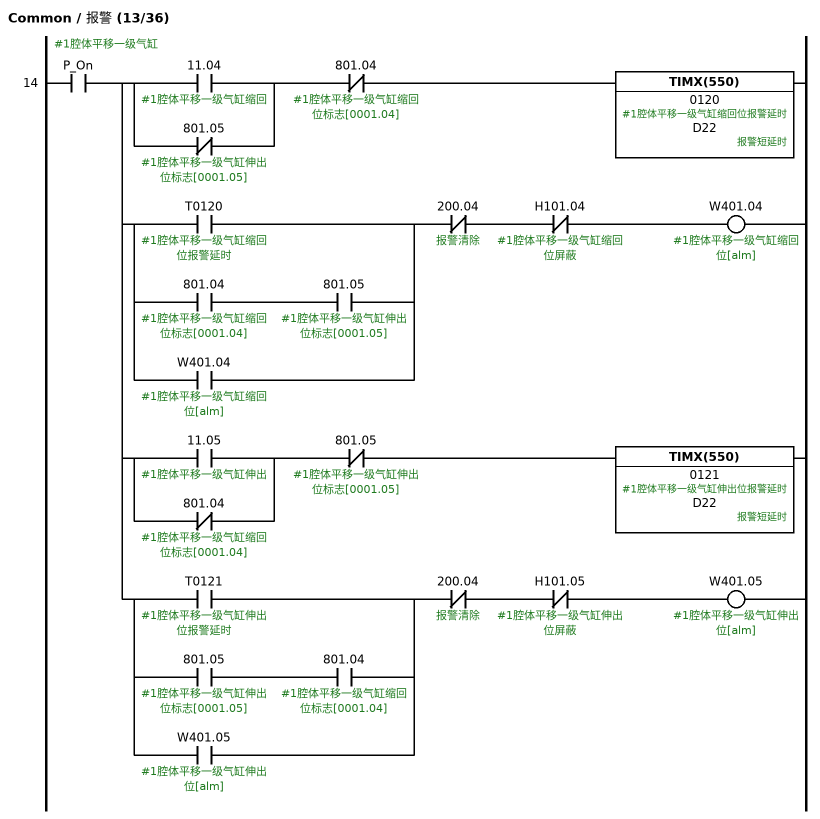
; [picture p528: Common / 报警, rungs 14-14]
; rung 14: #1腔体平移一级气缸
LD P_On
OUT TR0
LD 11.04  ; #1腔体平移一级气缸缩回
ORNOT 801.05  ; #1腔体平移一级气缸伸出位标志[0001.05]
ANDLD
ANDNOT 801.04  ; #1腔体平移一级气缸缩回位标志[0001.04]
TIMX(550) 0120 D22  ; 报警短延时, #1腔体平移一级气缸缩回位报警延时
LD TR0
LD T0120  ; #1腔体平移一级气缸缩回位报警延时
LD 801.04  ; #1腔体平移一级气缸缩回位标志[0001.04]
AND 801.05  ; #1腔体平移一级气缸伸出位标志[0001.05]
ORLD
OR W401.04  ; #1腔体平移一级气缸缩回位[alm]
ANDLD
ANDNOT 200.04  ; 报警清除
ANDNOT H101.04  ; #1腔体平移一级气缸缩回位屏蔽
OUT W401.04  ; #1腔体平移一级气缸缩回位[alm]
LD TR0
LD 11.05  ; #1腔体平移一级气缸伸出
ORNOT 801.04  ; #1腔体平移一级气缸缩回位标志[0001.04]
ANDLD
ANDNOT 801.05  ; #1腔体平移一级气缸伸出位标志[0001.05]
TIMX(550) 0121 D22  ; 报警短延时, #1腔体平移一级气缸伸出位报警延时
LD TR0
LD T0121  ; #1腔体平移一级气缸伸出位报警延时
LD 801.05  ; #1腔体平移一级气缸伸出位标志[0001.05]
AND 801.04  ; #1腔体平移一级气缸缩回位标志[0001.04]
ORLD
OR W401.05  ; #1腔体平移一级气缸伸出位[alm]
ANDLD
ANDNOT 200.04  ; 报警清除
ANDNOT H101.05  ; #1腔体平移一级气缸伸出位屏蔽
OUT W401.05  ; #1腔体平移一级气缸伸出位[alm]

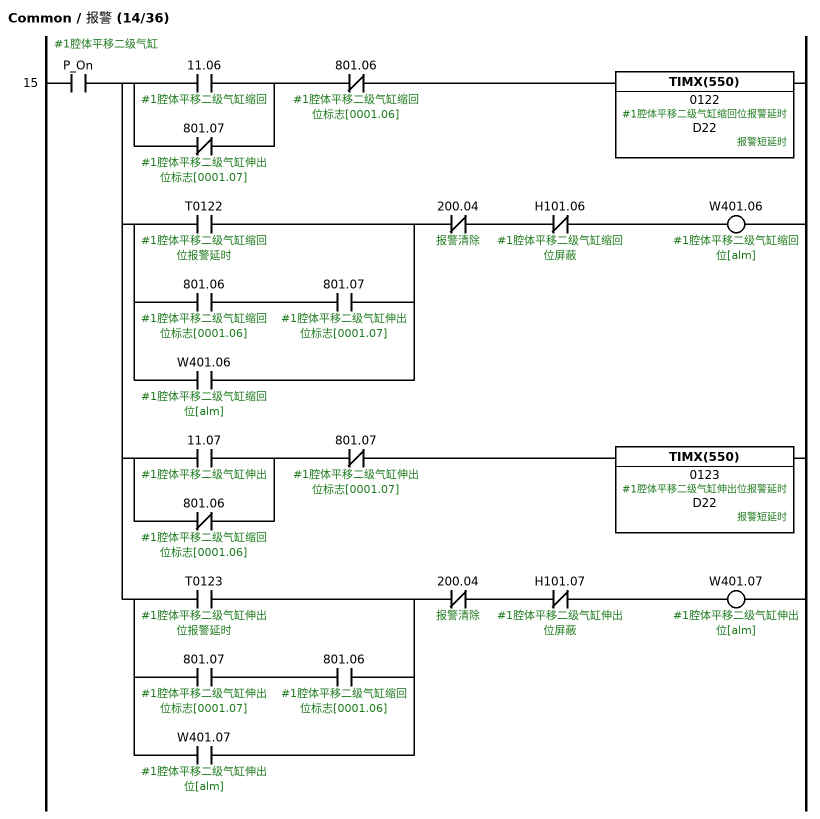
; rung 15: #1腔体平移二级气缸
LD P_On
OUT TR0
LD 11.06  ; #1腔体平移二级气缸缩回
ORNOT 801.07  ; #1腔体平移二级气缸伸出位标志[0001.07]
ANDLD
ANDNOT 801.06  ; #1腔体平移二级气缸缩回位标志[0001.06]
TIMX(550) 0122 D22  ; 报警短延时, #1腔体平移二级气缸缩回位报警延时
LD TR0
LD T0122  ; #1腔体平移二级气缸缩回位报警延时
LD 801.06  ; #1腔体平移二级气缸缩回位标志[0001.06]
AND 801.07  ; #1腔体平移二级气缸伸出位标志[0001.07]
ORLD
OR W401.06  ; #1腔体平移二级气缸缩回位[alm]
ANDLD
ANDNOT 200.04  ; 报警清除
ANDNOT H101.06  ; #1腔体平移二级气缸缩回位屏蔽
OUT W401.06  ; #1腔体平移二级气缸缩回位[alm]
LD TR0
LD 11.07  ; #1腔体平移二级气缸伸出
ORNOT 801.06  ; #1腔体平移二级气缸缩回位标志[0001.06]
ANDLD
ANDNOT 801.07  ; #1腔体平移二级气缸伸出位标志[0001.07]
TIMX(550) 0123 D22  ; 报警短延时, #1腔体平移二级气缸伸出位报警延时
LD TR0
LD T0123  ; #1腔体平移二级气缸伸出位报警延时
LD 801.07  ; #1腔体平移二级气缸伸出位标志[0001.07]
AND 801.06  ; #1腔体平移二级气缸缩回位标志[0001.06]
ORLD
OR W401.07  ; #1腔体平移二级气缸伸出位[alm]
ANDLD
ANDNOT 200.04  ; 报警清除
ANDNOT H101.07  ; #1腔体平移二级气缸伸出位屏蔽
OUT W401.07  ; #1腔体平移二级气缸伸出位[alm]

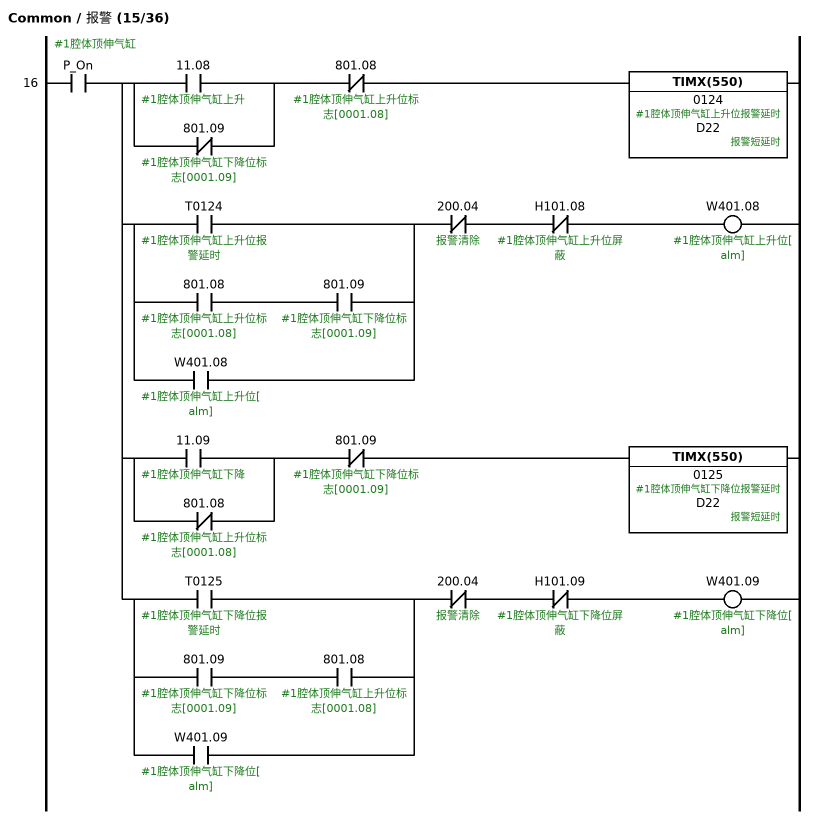
; rung 16: #1腔体顶伸气缸
LD P_On
OUT TR0
LD 11.08  ; #1腔体顶伸气缸上升
ORNOT 801.09  ; #1腔体顶伸气缸下降位标志[0001.09]
ANDLD
ANDNOT 801.08  ; #1腔体顶伸气缸上升位标志[0001.08]
TIMX(550) 0124 D22  ; 报警短延时, #1腔体顶伸气缸上升位报警延时
LD TR0
LD T0124  ; #1腔体顶伸气缸上升位报警延时
LD 801.08  ; #1腔体顶伸气缸上升位标志[0001.08]
AND 801.09  ; #1腔体顶伸气缸下降位标志[0001.09]
ORLD
OR W401.08  ; #1腔体顶伸气缸上升位[alm]
ANDLD
ANDNOT 200.04  ; 报警清除
ANDNOT H101.08  ; #1腔体顶伸气缸上升位屏蔽
OUT W401.08  ; #1腔体顶伸气缸上升位[alm]
LD TR0
LD 11.09  ; #1腔体顶伸气缸下降
ORNOT 801.08  ; #1腔体顶伸气缸上升位标志[0001.08]
ANDLD
ANDNOT 801.09  ; #1腔体顶伸气缸下降位标志[0001.09]
TIMX(550) 0125 D22  ; 报警短延时, #1腔体顶伸气缸下降位报警延时
LD TR0
LD T0125  ; #1腔体顶伸气缸下降位报警延时
LD 801.09  ; #1腔体顶伸气缸下降位标志[0001.09]
AND 801.08  ; #1腔体顶伸气缸上升位标志[0001.08]
ORLD
OR W401.09  ; #1腔体顶伸气缸下降位[alm]
ANDLD
ANDNOT 200.04  ; 报警清除
ANDNOT H101.09  ; #1腔体顶伸气缸下降位屏蔽
OUT W401.09  ; #1腔体顶伸气缸下降位[alm]

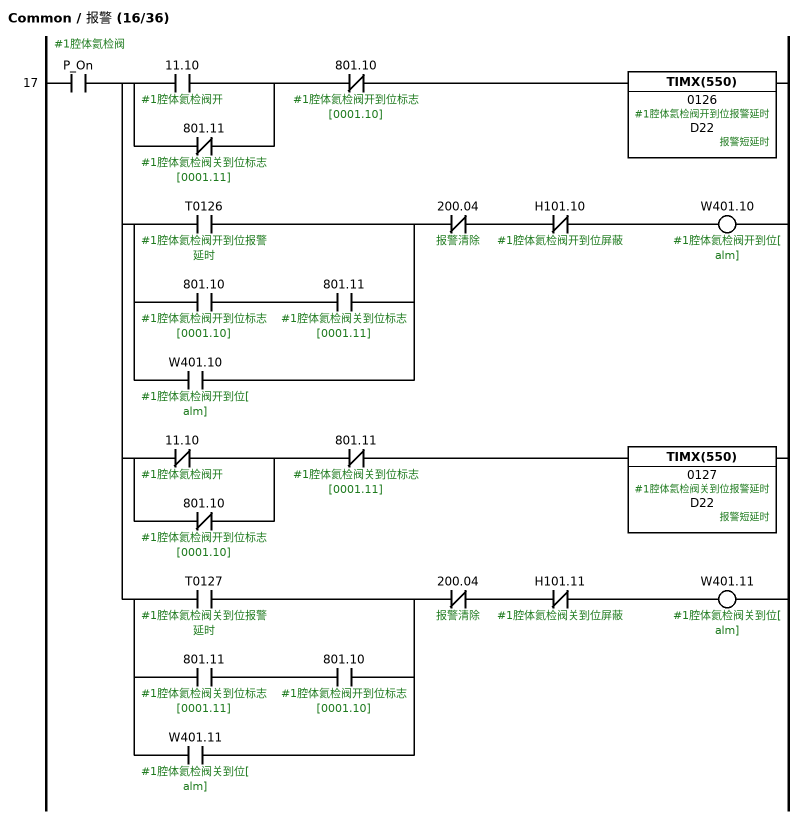
; rung 17: #1腔体氦检阀
LD P_On
OUT TR0
LD 11.10  ; #1腔体氦检阀开
ORNOT 801.11  ; #1腔体氦检阀关到位标志[0001.11]
ANDLD
ANDNOT 801.10  ; #1腔体氦检阀开到位标志[0001.10]
TIMX(550) 0126 D22  ; 报警短延时, #1腔体氦检阀开到位报警延时
LD TR0
LD T0126  ; #1腔体氦检阀开到位报警延时
LD 801.10  ; #1腔体氦检阀开到位标志[0001.10]
AND 801.11  ; #1腔体氦检阀关到位标志[0001.11]
ORLD
OR W401.10  ; #1腔体氦检阀开到位[alm]
ANDLD
ANDNOT 200.04  ; 报警清除
ANDNOT H101.10  ; #1腔体氦检阀开到位屏蔽
OUT W401.10  ; #1腔体氦检阀开到位[alm]
LD TR0
LDNOT 11.10  ; #1腔体氦检阀开
ORNOT 801.10  ; #1腔体氦检阀开到位标志[0001.10]
ANDLD
ANDNOT 801.11  ; #1腔体氦检阀关到位标志[0001.11]
TIMX(550) 0127 D22  ; 报警短延时, #1腔体氦检阀关到位报警延时
LD TR0
LD T0127  ; #1腔体氦检阀关到位报警延时
LD 801.11  ; #1腔体氦检阀关到位标志[0001.11]
AND 801.10  ; #1腔体氦检阀开到位标志[0001.10]
ORLD
OR W401.11  ; #1腔体氦检阀关到位[alm]
ANDLD
ANDNOT 200.04  ; 报警清除
ANDNOT H101.11  ; #1腔体氦检阀关到位屏蔽
OUT W401.11  ; #1腔体氦检阀关到位[alm]

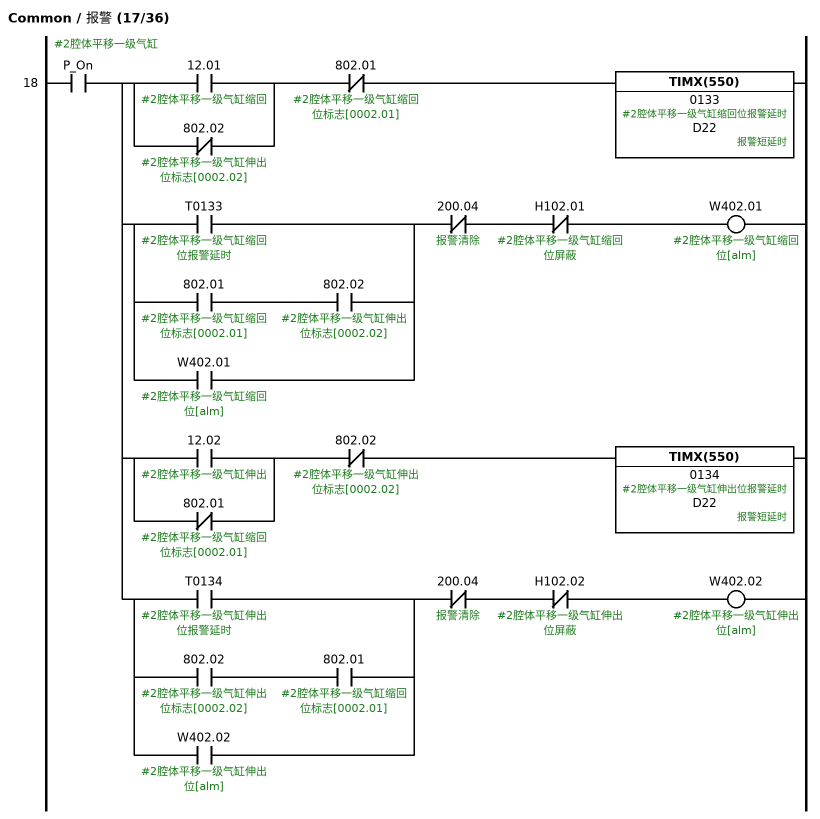
; rung 18: #2腔体平移一级气缸
LD P_On
OUT TR0
LD 12.01  ; #2腔体平移一级气缸缩回
ORNOT 802.02  ; #2腔体平移一级气缸伸出位标志[0002.02]
ANDLD
ANDNOT 802.01  ; #2腔体平移一级气缸缩回位标志[0002.01]
TIMX(550) 0133 D22  ; 报警短延时, #2腔体平移一级气缸缩回位报警延时
LD TR0
LD T0133  ; #2腔体平移一级气缸缩回位报警延时
LD 802.01  ; #2腔体平移一级气缸缩回位标志[0002.01]
AND 802.02  ; #2腔体平移一级气缸伸出位标志[0002.02]
ORLD
OR W402.01  ; #2腔体平移一级气缸缩回位[alm]
ANDLD
ANDNOT 200.04  ; 报警清除
ANDNOT H102.01  ; #2腔体平移一级气缸缩回位屏蔽
OUT W402.01  ; #2腔体平移一级气缸缩回位[alm]
LD TR0
LD 12.02  ; #2腔体平移一级气缸伸出
ORNOT 802.01  ; #2腔体平移一级气缸缩回位标志[0002.01]
ANDLD
ANDNOT 802.02  ; #2腔体平移一级气缸伸出位标志[0002.02]
TIMX(550) 0134 D22  ; 报警短延时, #2腔体平移一级气缸伸出位报警延时
LD TR0
LD T0134  ; #2腔体平移一级气缸伸出位报警延时
LD 802.02  ; #2腔体平移一级气缸伸出位标志[0002.02]
AND 802.01  ; #2腔体平移一级气缸缩回位标志[0002.01]
ORLD
OR W402.02  ; #2腔体平移一级气缸伸出位[alm]
ANDLD
ANDNOT 200.04  ; 报警清除
ANDNOT H102.02  ; #2腔体平移一级气缸伸出位屏蔽
OUT W402.02  ; #2腔体平移一级气缸伸出位[alm]

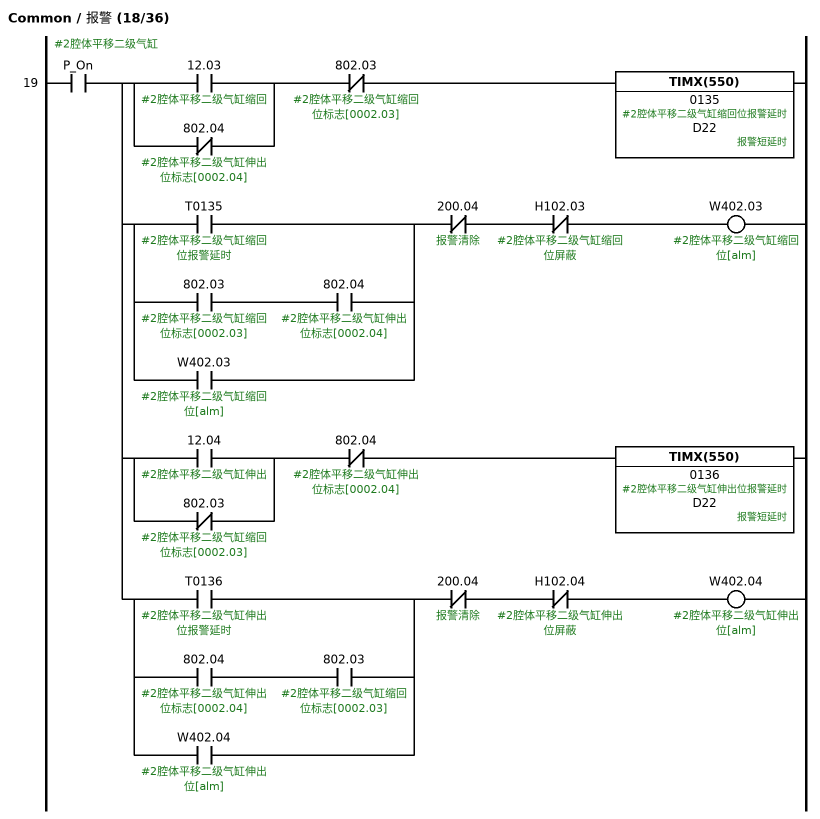
; rung 19: #2腔体平移二级气缸
LD P_On
OUT TR0
LD 12.03  ; #2腔体平移二级气缸缩回
ORNOT 802.04  ; #2腔体平移二级气缸伸出位标志[0002.04]
ANDLD
ANDNOT 802.03  ; #2腔体平移二级气缸缩回位标志[0002.03]
TIMX(550) 0135 D22  ; 报警短延时, #2腔体平移二级气缸缩回位报警延时
LD TR0
LD T0135  ; #2腔体平移二级气缸缩回位报警延时
LD 802.03  ; #2腔体平移二级气缸缩回位标志[0002.03]
AND 802.04  ; #2腔体平移二级气缸伸出位标志[0002.04]
ORLD
OR W402.03  ; #2腔体平移二级气缸缩回位[alm]
ANDLD
ANDNOT 200.04  ; 报警清除
ANDNOT H102.03  ; #2腔体平移二级气缸缩回位屏蔽
OUT W402.03  ; #2腔体平移二级气缸缩回位[alm]
LD TR0
LD 12.04  ; #2腔体平移二级气缸伸出
ORNOT 802.03  ; #2腔体平移二级气缸缩回位标志[0002.03]
ANDLD
ANDNOT 802.04  ; #2腔体平移二级气缸伸出位标志[0002.04]
TIMX(550) 0136 D22  ; 报警短延时, #2腔体平移二级气缸伸出位报警延时
LD TR0
LD T0136  ; #2腔体平移二级气缸伸出位报警延时
LD 802.04  ; #2腔体平移二级气缸伸出位标志[0002.04]
AND 802.03  ; #2腔体平移二级气缸缩回位标志[0002.03]
ORLD
OR W402.04  ; #2腔体平移二级气缸伸出位[alm]
ANDLD
ANDNOT 200.04  ; 报警清除
ANDNOT H102.04  ; #2腔体平移二级气缸伸出位屏蔽
OUT W402.04  ; #2腔体平移二级气缸伸出位[alm]

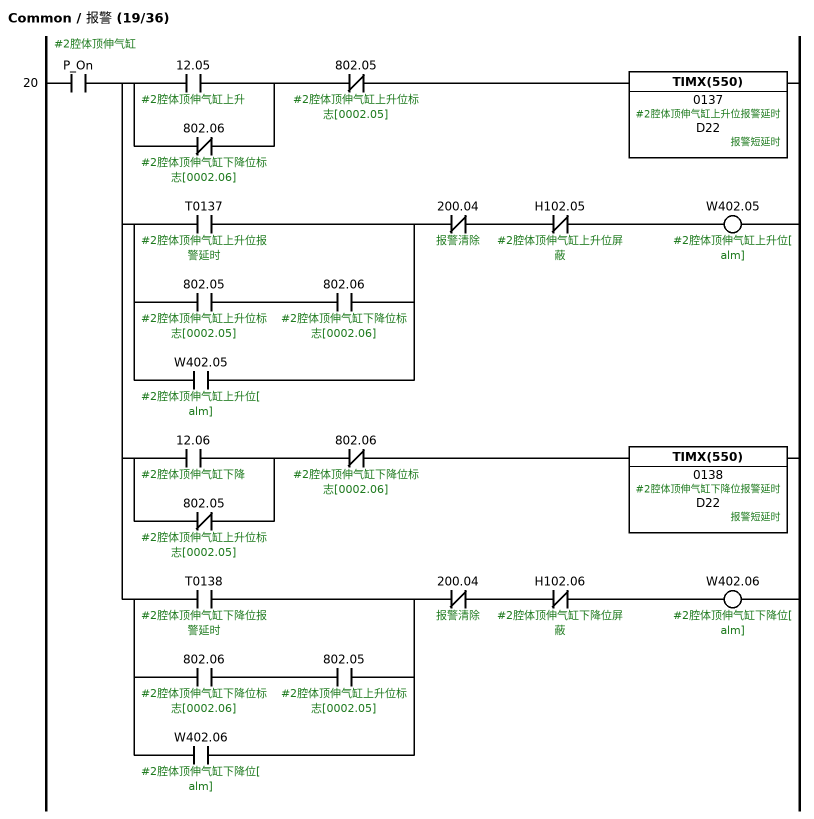
; rung 20: #2腔体顶伸气缸
LD P_On
OUT TR0
LD 12.05  ; #2腔体顶伸气缸上升
ORNOT 802.06  ; #2腔体顶伸气缸下降位标志[0002.06]
ANDLD
ANDNOT 802.05  ; #2腔体顶伸气缸上升位标志[0002.05]
TIMX(550) 0137 D22  ; 报警短延时, #2腔体顶伸气缸上升位报警延时
LD TR0
LD T0137  ; #2腔体顶伸气缸上升位报警延时
LD 802.05  ; #2腔体顶伸气缸上升位标志[0002.05]
AND 802.06  ; #2腔体顶伸气缸下降位标志[0002.06]
ORLD
OR W402.05  ; #2腔体顶伸气缸上升位[alm]
ANDLD
ANDNOT 200.04  ; 报警清除
ANDNOT H102.05  ; #2腔体顶伸气缸上升位屏蔽
OUT W402.05  ; #2腔体顶伸气缸上升位[alm]
LD TR0
LD 12.06  ; #2腔体顶伸气缸下降
ORNOT 802.05  ; #2腔体顶伸气缸上升位标志[0002.05]
ANDLD
ANDNOT 802.06  ; #2腔体顶伸气缸下降位标志[0002.06]
TIMX(550) 0138 D22  ; 报警短延时, #2腔体顶伸气缸下降位报警延时
LD TR0
LD T0138  ; #2腔体顶伸气缸下降位报警延时
LD 802.06  ; #2腔体顶伸气缸下降位标志[0002.06]
AND 802.05  ; #2腔体顶伸气缸上升位标志[0002.05]
ORLD
OR W402.06  ; #2腔体顶伸气缸下降位[alm]
ANDLD
ANDNOT 200.04  ; 报警清除
ANDNOT H102.06  ; #2腔体顶伸气缸下降位屏蔽
OUT W402.06  ; #2腔体顶伸气缸下降位[alm]

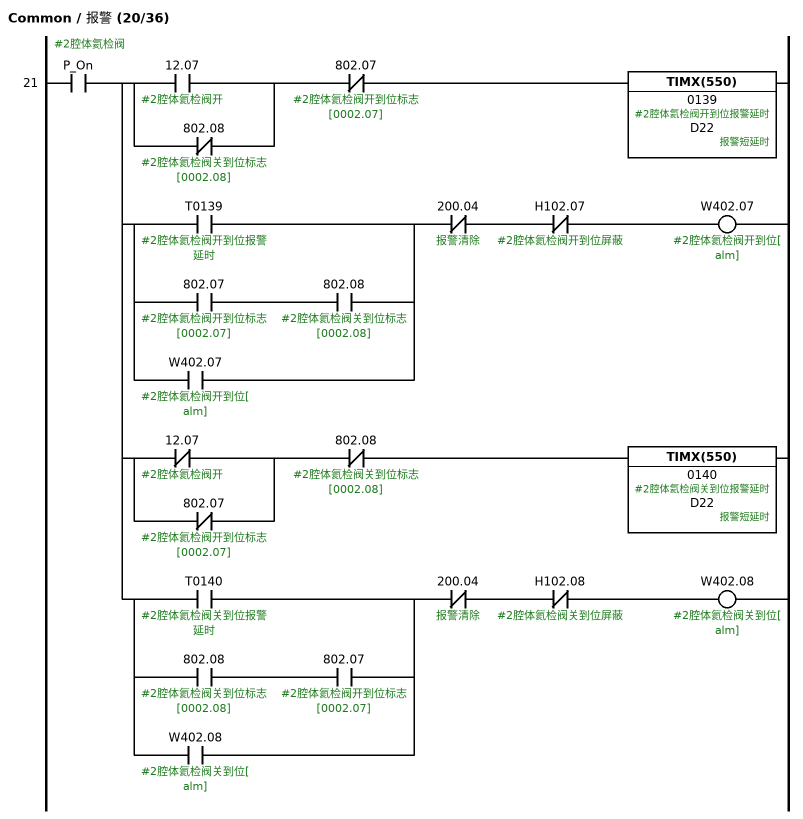
; rung 21: #2腔体氦检阀
LD P_On
OUT TR0
LD 12.07  ; #2腔体氦检阀开
ORNOT 802.08  ; #2腔体氦检阀关到位标志[0002.08]
ANDLD
ANDNOT 802.07  ; #2腔体氦检阀开到位标志[0002.07]
TIMX(550) 0139 D22  ; 报警短延时, #2腔体氦检阀开到位报警延时
LD TR0
LD T0139  ; #2腔体氦检阀开到位报警延时
LD 802.07  ; #2腔体氦检阀开到位标志[0002.07]
AND 802.08  ; #2腔体氦检阀关到位标志[0002.08]
ORLD
OR W402.07  ; #2腔体氦检阀开到位[alm]
ANDLD
ANDNOT 200.04  ; 报警清除
ANDNOT H102.07  ; #2腔体氦检阀开到位屏蔽
OUT W402.07  ; #2腔体氦检阀开到位[alm]
LD TR0
LDNOT 12.07  ; #2腔体氦检阀开
ORNOT 802.07  ; #2腔体氦检阀开到位标志[0002.07]
ANDLD
ANDNOT 802.08  ; #2腔体氦检阀关到位标志[0002.08]
TIMX(550) 0140 D22  ; 报警短延时, #2腔体氦检阀关到位报警延时
LD TR0
LD T0140  ; #2腔体氦检阀关到位报警延时
LD 802.08  ; #2腔体氦检阀关到位标志[0002.08]
AND 802.07  ; #2腔体氦检阀开到位标志[0002.07]
ORLD
OR W402.08  ; #2腔体氦检阀关到位[alm]
ANDLD
ANDNOT 200.04  ; 报警清除
ANDNOT H102.08  ; #2腔体氦检阀关到位屏蔽
OUT W402.08  ; #2腔体氦检阀关到位[alm]

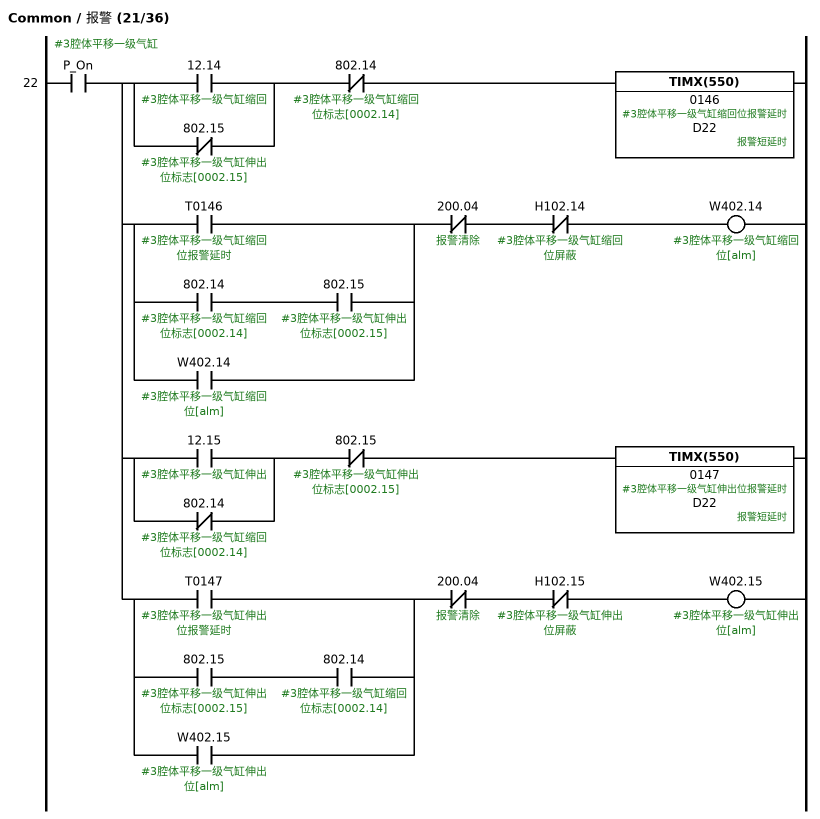
; rung 22: #3腔体平移一级气缸
LD P_On
OUT TR0
LD 12.14  ; #3腔体平移一级气缸缩回
ORNOT 802.15  ; #3腔体平移一级气缸伸出位标志[0002.15]
ANDLD
ANDNOT 802.14  ; #3腔体平移一级气缸缩回位标志[0002.14]
TIMX(550) 0146 D22  ; 报警短延时, #3腔体平移一级气缸缩回位报警延时
LD TR0
LD T0146  ; #3腔体平移一级气缸缩回位报警延时
LD 802.14  ; #3腔体平移一级气缸缩回位标志[0002.14]
AND 802.15  ; #3腔体平移一级气缸伸出位标志[0002.15]
ORLD
OR W402.14  ; #3腔体平移一级气缸缩回位[alm]
ANDLD
ANDNOT 200.04  ; 报警清除
ANDNOT H102.14  ; #3腔体平移一级气缸缩回位屏蔽
OUT W402.14  ; #3腔体平移一级气缸缩回位[alm]
LD TR0
LD 12.15  ; #3腔体平移一级气缸伸出
ORNOT 802.14  ; #3腔体平移一级气缸缩回位标志[0002.14]
ANDLD
ANDNOT 802.15  ; #3腔体平移一级气缸伸出位标志[0002.15]
TIMX(550) 0147 D22  ; 报警短延时, #3腔体平移一级气缸伸出位报警延时
LD TR0
LD T0147  ; #3腔体平移一级气缸伸出位报警延时
LD 802.15  ; #3腔体平移一级气缸伸出位标志[0002.15]
AND 802.14  ; #3腔体平移一级气缸缩回位标志[0002.14]
ORLD
OR W402.15  ; #3腔体平移一级气缸伸出位[alm]
ANDLD
ANDNOT 200.04  ; 报警清除
ANDNOT H102.15  ; #3腔体平移一级气缸伸出位屏蔽
OUT W402.15  ; #3腔体平移一级气缸伸出位[alm]

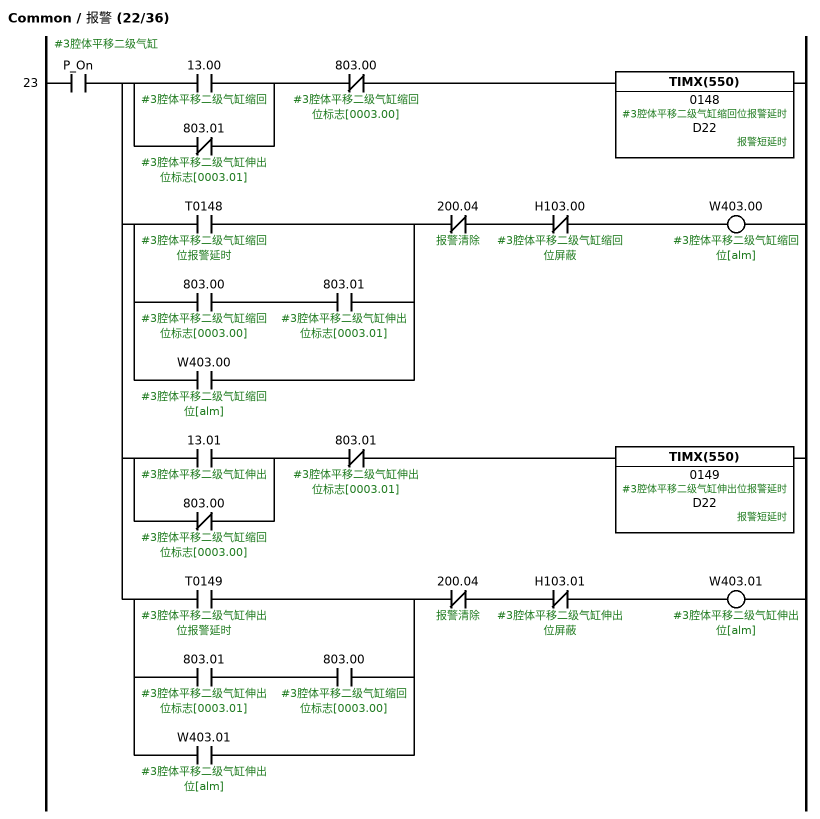
; rung 23: #3腔体平移二级气缸
LD P_On
OUT TR0
LD 13.00  ; #3腔体平移二级气缸缩回
ORNOT 803.01  ; #3腔体平移二级气缸伸出位标志[0003.01]
ANDLD
ANDNOT 803.00  ; #3腔体平移二级气缸缩回位标志[0003.00]
TIMX(550) 0148 D22  ; 报警短延时, #3腔体平移二级气缸缩回位报警延时
LD TR0
LD T0148  ; #3腔体平移二级气缸缩回位报警延时
LD 803.00  ; #3腔体平移二级气缸缩回位标志[0003.00]
AND 803.01  ; #3腔体平移二级气缸伸出位标志[0003.01]
ORLD
OR W403.00  ; #3腔体平移二级气缸缩回位[alm]
ANDLD
ANDNOT 200.04  ; 报警清除
ANDNOT H103.00  ; #3腔体平移二级气缸缩回位屏蔽
OUT W403.00  ; #3腔体平移二级气缸缩回位[alm]
LD TR0
LD 13.01  ; #3腔体平移二级气缸伸出
ORNOT 803.00  ; #3腔体平移二级气缸缩回位标志[0003.00]
ANDLD
ANDNOT 803.01  ; #3腔体平移二级气缸伸出位标志[0003.01]
TIMX(550) 0149 D22  ; 报警短延时, #3腔体平移二级气缸伸出位报警延时
LD TR0
LD T0149  ; #3腔体平移二级气缸伸出位报警延时
LD 803.01  ; #3腔体平移二级气缸伸出位标志[0003.01]
AND 803.00  ; #3腔体平移二级气缸缩回位标志[0003.00]
ORLD
OR W403.01  ; #3腔体平移二级气缸伸出位[alm]
ANDLD
ANDNOT 200.04  ; 报警清除
ANDNOT H103.01  ; #3腔体平移二级气缸伸出位屏蔽
OUT W403.01  ; #3腔体平移二级气缸伸出位[alm]

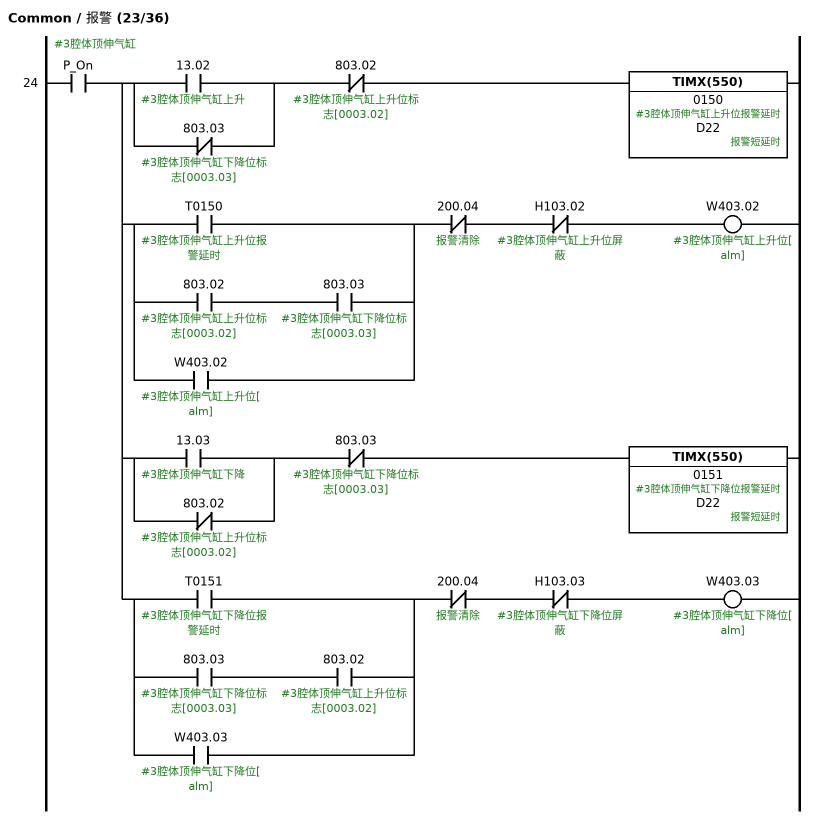
; rung 24: #3腔体顶伸气缸
LD P_On
OUT TR0
LD 13.02  ; #3腔体顶伸气缸上升
ORNOT 803.03  ; #3腔体顶伸气缸下降位标志[0003.03]
ANDLD
ANDNOT 803.02  ; #3腔体顶伸气缸上升位标志[0003.02]
TIMX(550) 0150 D22  ; 报警短延时, #3腔体顶伸气缸上升位报警延时
LD TR0
LD T0150  ; #3腔体顶伸气缸上升位报警延时
LD 803.02  ; #3腔体顶伸气缸上升位标志[0003.02]
AND 803.03  ; #3腔体顶伸气缸下降位标志[0003.03]
ORLD
OR W403.02  ; #3腔体顶伸气缸上升位[alm]
ANDLD
ANDNOT 200.04  ; 报警清除
ANDNOT H103.02  ; #3腔体顶伸气缸上升位屏蔽
OUT W403.02  ; #3腔体顶伸气缸上升位[alm]
LD TR0
LD 13.03  ; #3腔体顶伸气缸下降
ORNOT 803.02  ; #3腔体顶伸气缸上升位标志[0003.02]
ANDLD
ANDNOT 803.03  ; #3腔体顶伸气缸下降位标志[0003.03]
TIMX(550) 0151 D22  ; 报警短延时, #3腔体顶伸气缸下降位报警延时
LD TR0
LD T0151  ; #3腔体顶伸气缸下降位报警延时
LD 803.03  ; #3腔体顶伸气缸下降位标志[0003.03]
AND 803.02  ; #3腔体顶伸气缸上升位标志[0003.02]
ORLD
OR W403.03  ; #3腔体顶伸气缸下降位[alm]
ANDLD
ANDNOT 200.04  ; 报警清除
ANDNOT H103.03  ; #3腔体顶伸气缸下降位屏蔽
OUT W403.03  ; #3腔体顶伸气缸下降位[alm]

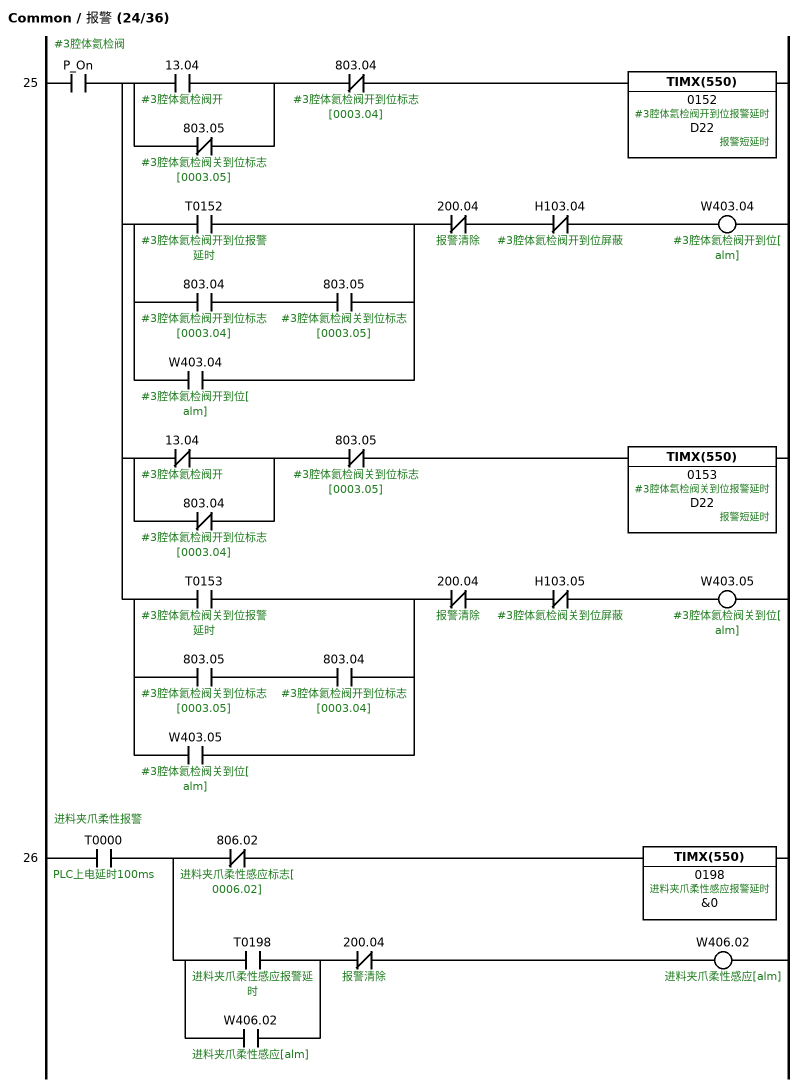
; rung 25: #3腔体氦检阀
LD P_On
OUT TR0
LD 13.04  ; #3腔体氦检阀开
ORNOT 803.05  ; #3腔体氦检阀关到位标志[0003.05]
ANDLD
ANDNOT 803.04  ; #3腔体氦检阀开到位标志[0003.04]
TIMX(550) 0152 D22  ; 报警短延时, #3腔体氦检阀开到位报警延时
LD TR0
LD T0152  ; #3腔体氦检阀开到位报警延时
LD 803.04  ; #3腔体氦检阀开到位标志[0003.04]
AND 803.05  ; #3腔体氦检阀关到位标志[0003.05]
ORLD
OR W403.04  ; #3腔体氦检阀开到位[alm]
ANDLD
ANDNOT 200.04  ; 报警清除
ANDNOT H103.04  ; #3腔体氦检阀开到位屏蔽
OUT W403.04  ; #3腔体氦检阀开到位[alm]
LD TR0
LDNOT 13.04  ; #3腔体氦检阀开
ORNOT 803.04  ; #3腔体氦检阀开到位标志[0003.04]
ANDLD
ANDNOT 803.05  ; #3腔体氦检阀关到位标志[0003.05]
TIMX(550) 0153 D22  ; 报警短延时, #3腔体氦检阀关到位报警延时
LD TR0
LD T0153  ; #3腔体氦检阀关到位报警延时
LD 803.05  ; #3腔体氦检阀关到位标志[0003.05]
AND 803.04  ; #3腔体氦检阀开到位标志[0003.04]
ORLD
OR W403.05  ; #3腔体氦检阀关到位[alm]
ANDLD
ANDNOT 200.04  ; 报警清除
ANDNOT H103.05  ; #3腔体氦检阀关到位屏蔽
OUT W403.05  ; #3腔体氦检阀关到位[alm]
; rung 26: 进料夹爪柔性报警
LD T0000  ; PLC上电延时100ms
OUT TR0
ANDNOT 806.02  ; 进料夹爪柔性感应标志[0006.02]
TIMX(550) 0198 &0  ; 进料夹爪柔性感应报警延时
LD TR0
LD T0198  ; 进料夹爪柔性感应报警延时
OR W406.02  ; 进料夹爪柔性感应[alm]
ANDLD
ANDNOT 200.04  ; 报警清除
OUT W406.02  ; 进料夹爪柔性感应[alm]

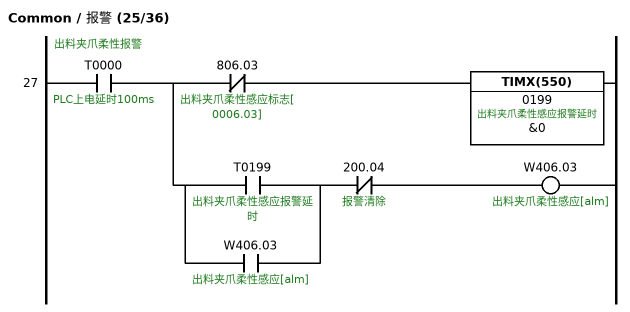
; rung 27: 出料夹爪柔性报警
LD T0000  ; PLC上电延时100ms
OUT TR0
ANDNOT 806.03  ; 出料夹爪柔性感应标志[0006.03]
TIMX(550) 0199 &0  ; 出料夹爪柔性感应报警延时
LD TR0
LD T0199  ; 出料夹爪柔性感应报警延时
OR W406.03  ; 出料夹爪柔性感应[alm]
ANDLD
ANDNOT 200.04  ; 报警清除
OUT W406.03  ; 出料夹爪柔性感应[alm]

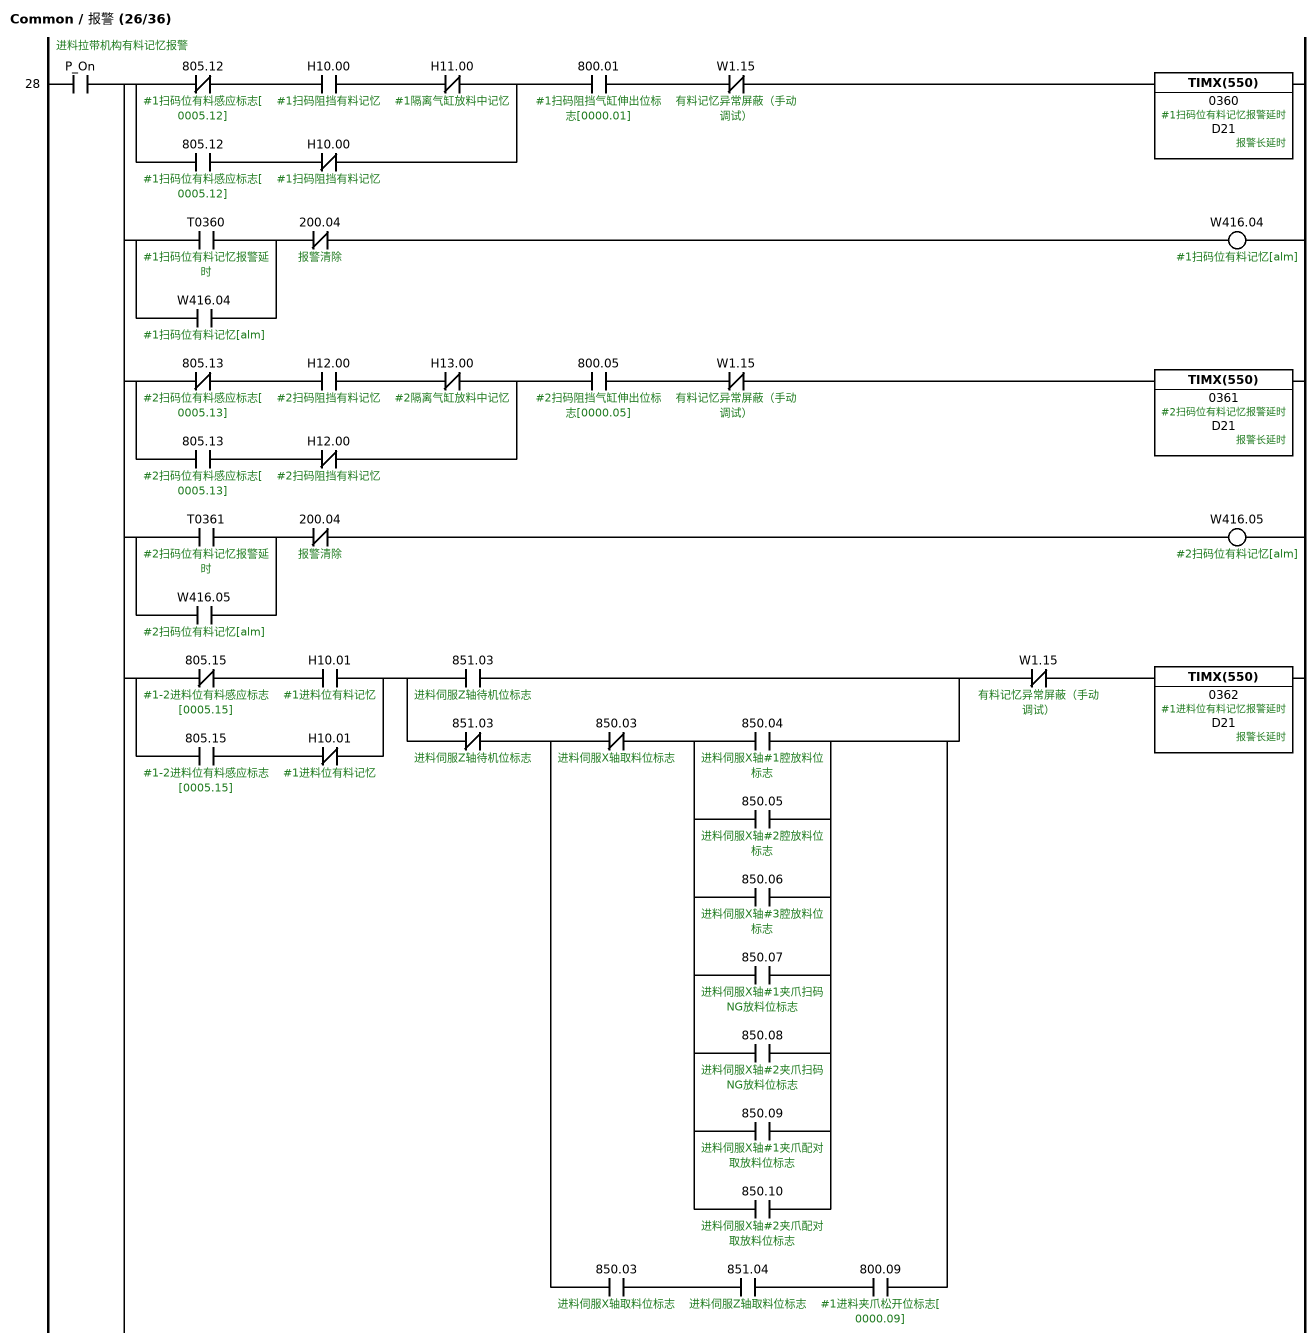

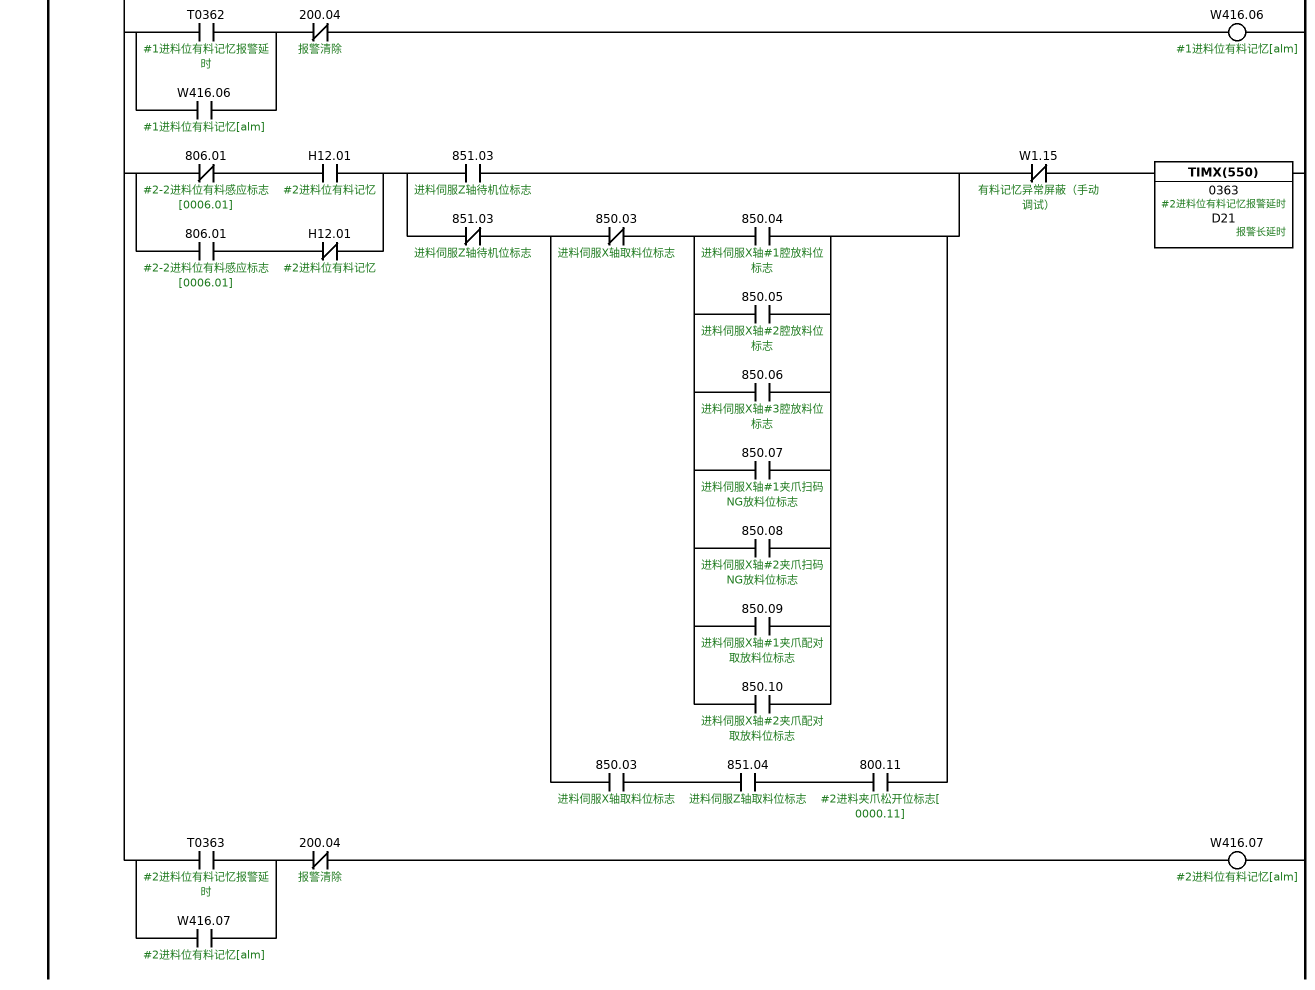
; rung 28: 进料拉带机构有料记忆报警
LD P_On
OUT TR0
LDNOT 805.12  ; #1扫码位有料感应标志[0005.12]
AND H10.00  ; #1扫码阻挡有料记忆
ANDNOT H11.00  ; #1隔离气缸放料中记忆
LD 805.12  ; #1扫码位有料感应标志[0005.12]
ANDNOT H10.00  ; #1扫码阻挡有料记忆
ORLD
ANDLD
AND 800.01  ; #1扫码阻挡气缸伸出位标志[0000.01]
ANDNOT W1.15  ; 有料记忆异常屏蔽（手动调试）
TIMX(550) 0360 D21  ; 报警长延时, #1扫码位有料记忆报警延时
LD TR0
LD T0360  ; #1扫码位有料记忆报警延时
OR W416.04  ; #1扫码位有料记忆[alm]
ANDLD
ANDNOT 200.04  ; 报警清除
OUT W416.04  ; #1扫码位有料记忆[alm]
LD TR0
LDNOT 805.13  ; #2扫码位有料感应标志[0005.13]
AND H12.00  ; #2扫码阻挡有料记忆
ANDNOT H13.00  ; #2隔离气缸放料中记忆
LD 805.13  ; #2扫码位有料感应标志[0005.13]
ANDNOT H12.00  ; #2扫码阻挡有料记忆
ORLD
ANDLD
AND 800.05  ; #2扫码阻挡气缸伸出位标志[0000.05]
ANDNOT W1.15  ; 有料记忆异常屏蔽（手动调试）
TIMX(550) 0361 D21  ; 报警长延时, #2扫码位有料记忆报警延时
LD TR0
LD T0361  ; #2扫码位有料记忆报警延时
OR W416.05  ; #2扫码位有料记忆[alm]
ANDLD
ANDNOT 200.04  ; 报警清除
OUT W416.05  ; #2扫码位有料记忆[alm]
LD TR0
LDNOT 805.15  ; #1-2进料位有料感应标志[0005.15]
AND H10.01  ; #1进料位有料记忆
LD 805.15  ; #1-2进料位有料感应标志[0005.15]
ANDNOT H10.01  ; #1进料位有料记忆
ORLD
ANDLD
LD 851.03  ; 进料伺服Z轴待机位标志
LDNOT 851.03  ; 进料伺服Z轴待机位标志
LDNOT 850.03  ; 进料伺服X轴取料位标志
LD 850.04  ; 进料伺服X轴#1腔放料位标志
OR 850.05  ; 进料伺服X轴#2腔放料位标志
OR 850.06  ; 进料伺服X轴#3腔放料位标志
OR 850.07  ; 进料伺服X轴#1夹爪扫码NG放料位标志
OR 850.08  ; 进料伺服X轴#2夹爪扫码NG放料位标志
OR 850.09  ; 进料伺服X轴#1夹爪配对取放料位标志
OR 850.10  ; 进料伺服X轴#2夹爪配对取放料位标志
ANDLD
LD 850.03  ; 进料伺服X轴取料位标志
AND 851.04  ; 进料伺服Z轴取料位标志
AND 800.09  ; #1进料夹爪松开位标志[0000.09]
ORLD
ANDLD
ORLD
ANDLD
ANDNOT W1.15  ; 有料记忆异常屏蔽（手动调试）
TIMX(550) 0362 D21  ; 报警长延时, #1进料位有料记忆报警延时
LD TR0
LD T0362  ; #1进料位有料记忆报警延时
OR W416.06  ; #1进料位有料记忆[alm]
ANDLD
ANDNOT 200.04  ; 报警清除
OUT W416.06  ; #1进料位有料记忆[alm]
LD TR0
LDNOT 806.01  ; #2-2进料位有料感应标志[0006.01]
AND H12.01  ; #2进料位有料记忆
LD 806.01  ; #2-2进料位有料感应标志[0006.01]
ANDNOT H12.01  ; #2进料位有料记忆
ORLD
ANDLD
LD 851.03  ; 进料伺服Z轴待机位标志
LDNOT 851.03  ; 进料伺服Z轴待机位标志
LDNOT 850.03  ; 进料伺服X轴取料位标志
LD 850.04  ; 进料伺服X轴#1腔放料位标志
OR 850.05  ; 进料伺服X轴#2腔放料位标志
OR 850.06  ; 进料伺服X轴#3腔放料位标志
OR 850.07  ; 进料伺服X轴#1夹爪扫码NG放料位标志
OR 850.08  ; 进料伺服X轴#2夹爪扫码NG放料位标志
OR 850.09  ; 进料伺服X轴#1夹爪配对取放料位标志
OR 850.10  ; 进料伺服X轴#2夹爪配对取放料位标志
ANDLD
LD 850.03  ; 进料伺服X轴取料位标志
AND 851.04  ; 进料伺服Z轴取料位标志
AND 800.11  ; #2进料夹爪松开位标志[0000.11]
ORLD
ANDLD
ORLD
ANDLD
ANDNOT W1.15  ; 有料记忆异常屏蔽（手动调试）
TIMX(550) 0363 D21  ; 报警长延时, #2进料位有料记忆报警延时
LD TR0
LD T0363  ; #2进料位有料记忆报警延时
OR W416.07  ; #2进料位有料记忆[alm]
ANDLD
ANDNOT 200.04  ; 报警清除
OUT W416.07  ; #2进料位有料记忆[alm]

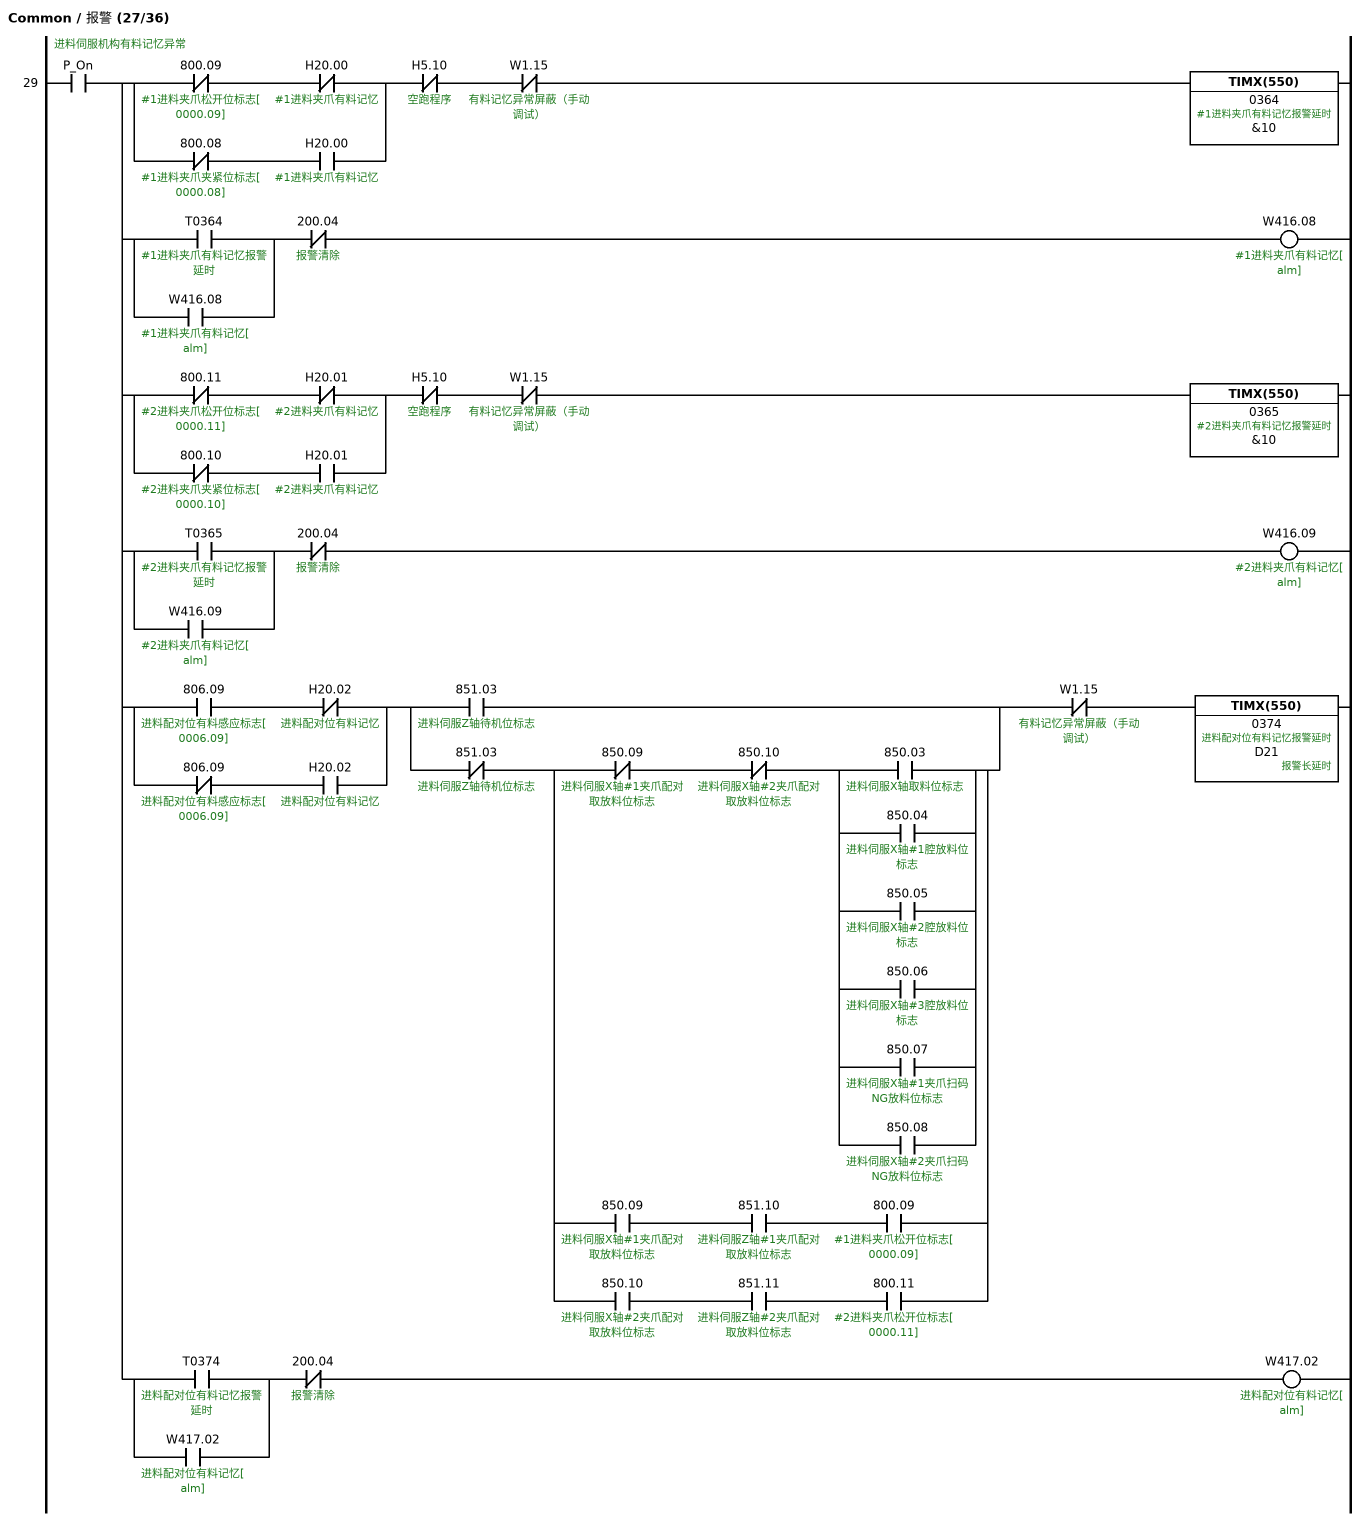
; rung 29: 进料伺服机构有料记忆异常
LD P_On
OUT TR0
LDNOT 800.09  ; #1进料夹爪松开位标志[0000.09]
ANDNOT H20.00  ; #1进料夹爪有料记忆
LDNOT 800.08  ; #1进料夹爪夹紧位标志[0000.08]
AND H20.00  ; #1进料夹爪有料记忆
ORLD
ANDLD
ANDNOT H5.10  ; 空跑程序
ANDNOT W1.15  ; 有料记忆异常屏蔽（手动调试）
TIMX(550) 0364 &10  ; #1进料夹爪有料记忆报警延时
LD TR0
LD T0364  ; #1进料夹爪有料记忆报警延时
OR W416.08  ; #1进料夹爪有料记忆[alm]
ANDLD
ANDNOT 200.04  ; 报警清除
OUT W416.08  ; #1进料夹爪有料记忆[alm]
LD TR0
LDNOT 800.11  ; #2进料夹爪松开位标志[0000.11]
ANDNOT H20.01  ; #2进料夹爪有料记忆
LDNOT 800.10  ; #2进料夹爪夹紧位标志[0000.10]
AND H20.01  ; #2进料夹爪有料记忆
ORLD
ANDLD
ANDNOT H5.10  ; 空跑程序
ANDNOT W1.15  ; 有料记忆异常屏蔽（手动调试）
TIMX(550) 0365 &10  ; #2进料夹爪有料记忆报警延时
LD TR0
LD T0365  ; #2进料夹爪有料记忆报警延时
OR W416.09  ; #2进料夹爪有料记忆[alm]
ANDLD
ANDNOT 200.04  ; 报警清除
OUT W416.09  ; #2进料夹爪有料记忆[alm]
LD TR0
LD 806.09  ; 进料配对位有料感应标志[0006.09]
ANDNOT H20.02  ; 进料配对位有料记忆
LDNOT 806.09  ; 进料配对位有料感应标志[0006.09]
AND H20.02  ; 进料配对位有料记忆
ORLD
ANDLD
LD 851.03  ; 进料伺服Z轴待机位标志
LDNOT 851.03  ; 进料伺服Z轴待机位标志
LDNOT 850.09  ; 进料伺服X轴#1夹爪配对取放料位标志
ANDNOT 850.10  ; 进料伺服X轴#2夹爪配对取放料位标志
LD 850.03  ; 进料伺服X轴取料位标志
OR 850.04  ; 进料伺服X轴#1腔放料位标志
OR 850.05  ; 进料伺服X轴#2腔放料位标志
OR 850.06  ; 进料伺服X轴#3腔放料位标志
OR 850.07  ; 进料伺服X轴#1夹爪扫码NG放料位标志
OR 850.08  ; 进料伺服X轴#2夹爪扫码NG放料位标志
ANDLD
LD 850.09  ; 进料伺服X轴#1夹爪配对取放料位标志
AND 851.10  ; 进料伺服Z轴#1夹爪配对取放料位标志
AND 800.09  ; #1进料夹爪松开位标志[0000.09]
ORLD
LD 850.10  ; 进料伺服X轴#2夹爪配对取放料位标志
AND 851.11  ; 进料伺服Z轴#2夹爪配对取放料位标志
AND 800.11  ; #2进料夹爪松开位标志[0000.11]
ORLD
ANDLD
ORLD
ANDLD
ANDNOT W1.15  ; 有料记忆异常屏蔽（手动调试）
TIMX(550) 0374 D21  ; 报警长延时, 进料配对位有料记忆报警延时
LD TR0
LD T0374  ; 进料配对位有料记忆报警延时
OR W417.02  ; 进料配对位有料记忆[alm]
ANDLD
ANDNOT 200.04  ; 报警清除
OUT W417.02  ; 进料配对位有料记忆[alm]

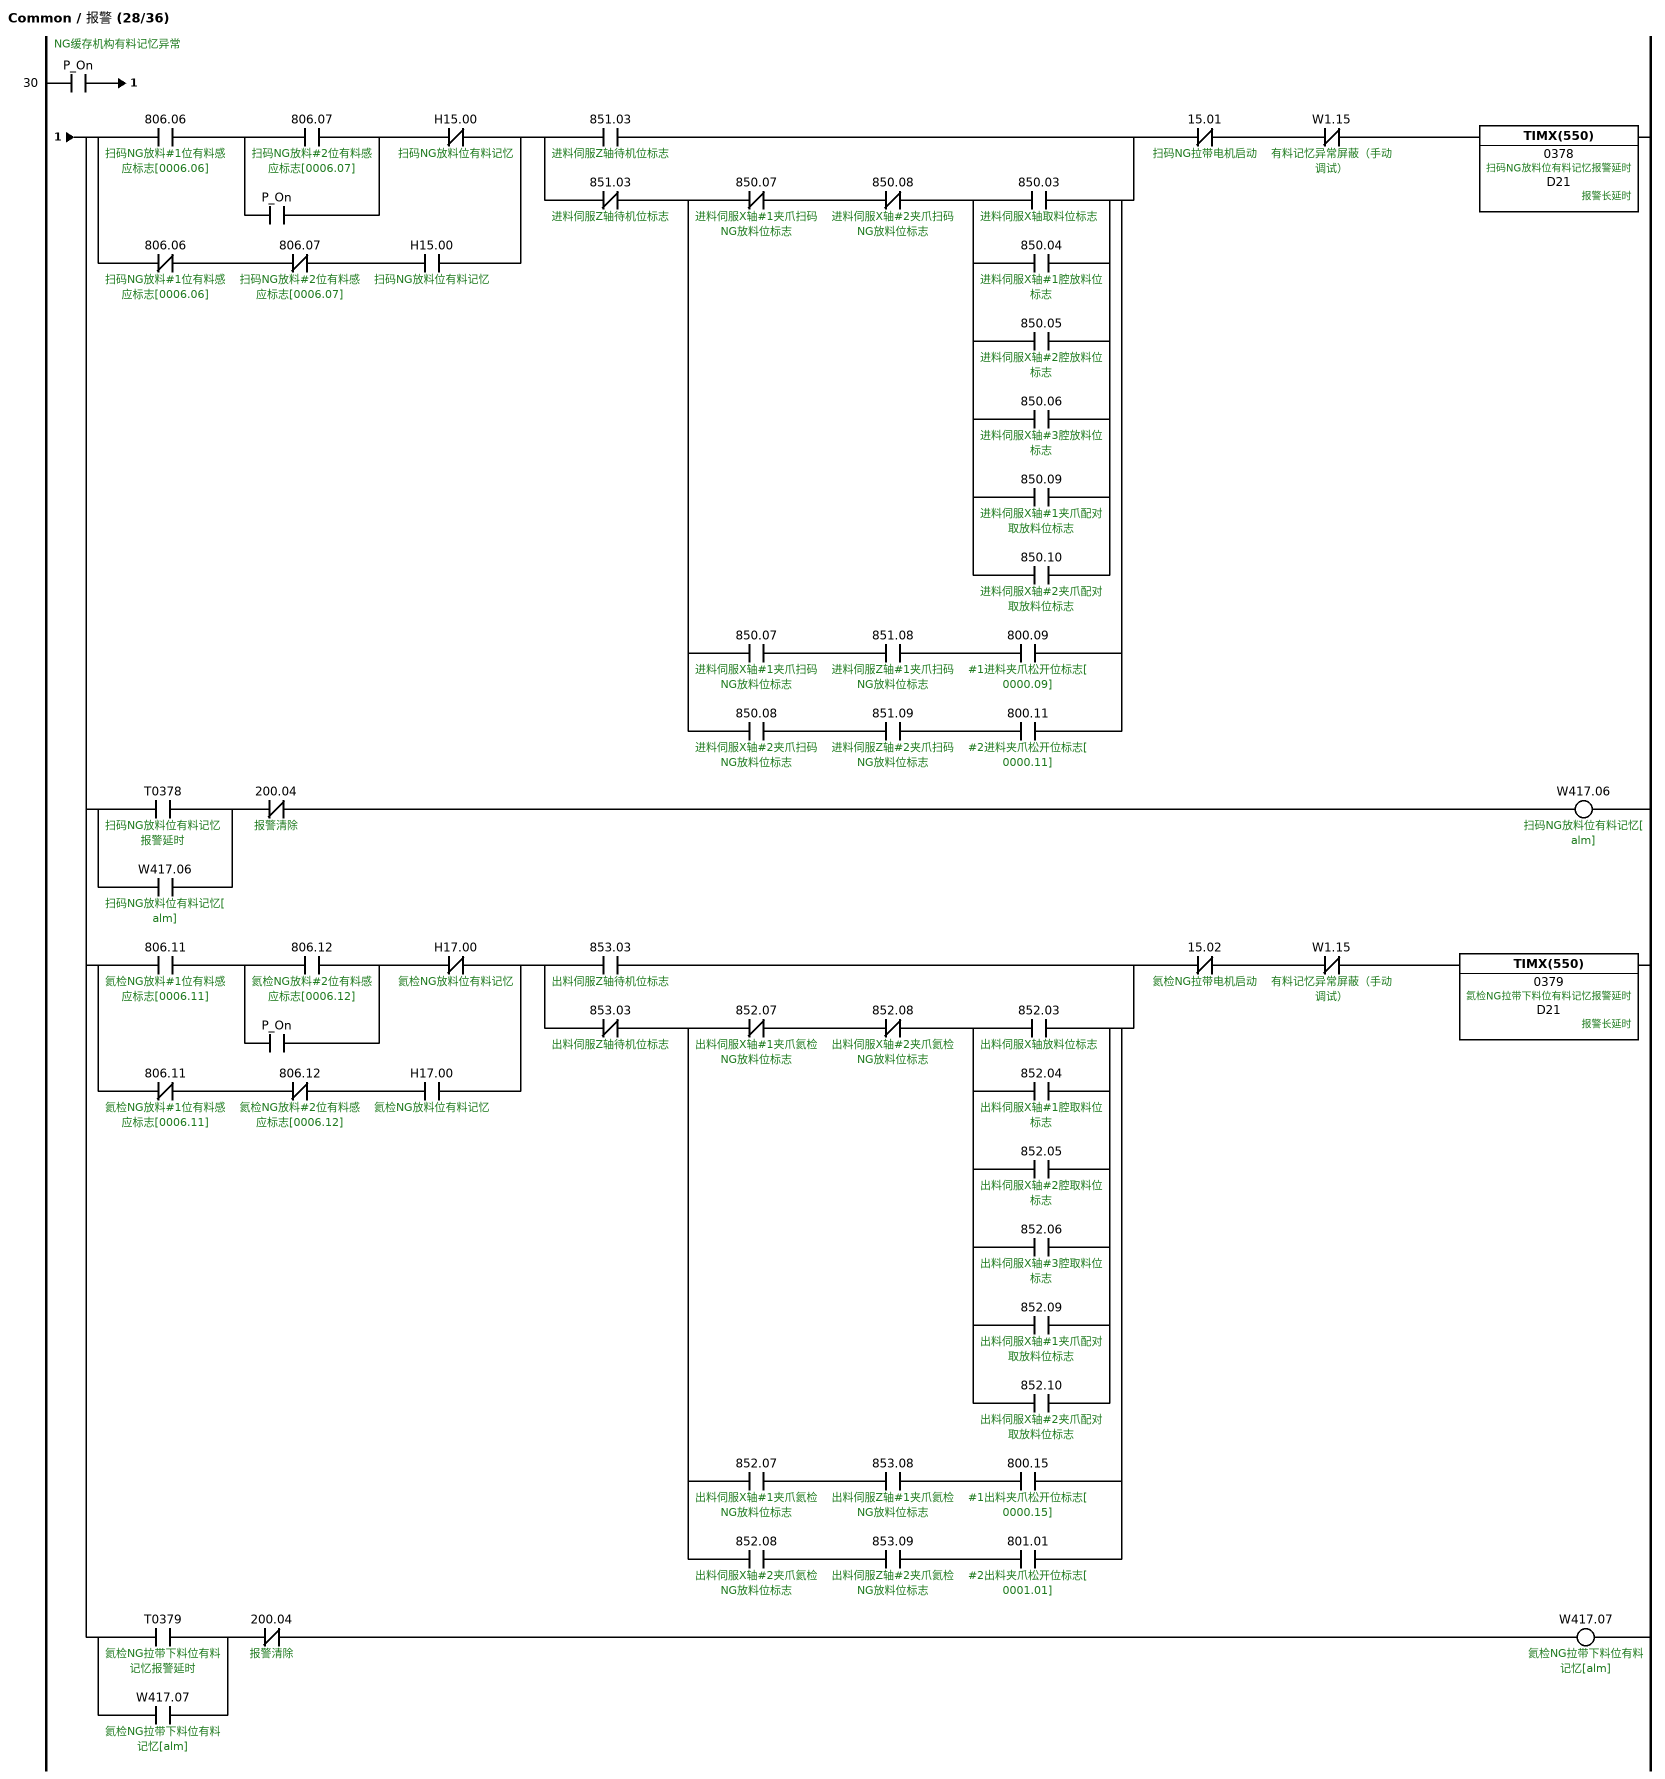
; rung 30: NG缓存机构有料记忆异常
LD P_On
OUT TR0
LD 806.06  ; 扫码NG放料#1位有料感应标志[0006.06]
LD 806.07  ; 扫码NG放料#2位有料感应标志[0006.07]
OR P_On
ANDLD
ANDNOT H15.00  ; 扫码NG放料位有料记忆
LDNOT 806.06  ; 扫码NG放料#1位有料感应标志[0006.06]
ANDNOT 806.07  ; 扫码NG放料#2位有料感应标志[0006.07]
AND H15.00  ; 扫码NG放料位有料记忆
ORLD
ANDLD
LD 851.03  ; 进料伺服Z轴待机位标志
LDNOT 851.03  ; 进料伺服Z轴待机位标志
LDNOT 850.07  ; 进料伺服X轴#1夹爪扫码NG放料位标志
ANDNOT 850.08  ; 进料伺服X轴#2夹爪扫码NG放料位标志
LD 850.03  ; 进料伺服X轴取料位标志
OR 850.04  ; 进料伺服X轴#1腔放料位标志
OR 850.05  ; 进料伺服X轴#2腔放料位标志
OR 850.06  ; 进料伺服X轴#3腔放料位标志
OR 850.09  ; 进料伺服X轴#1夹爪配对取放料位标志
OR 850.10  ; 进料伺服X轴#2夹爪配对取放料位标志
ANDLD
LD 850.07  ; 进料伺服X轴#1夹爪扫码NG放料位标志
AND 851.08  ; 进料伺服Z轴#1夹爪扫码NG放料位标志
AND 800.09  ; #1进料夹爪松开位标志[0000.09]
ORLD
LD 850.08  ; 进料伺服X轴#2夹爪扫码NG放料位标志
AND 851.09  ; 进料伺服Z轴#2夹爪扫码NG放料位标志
AND 800.11  ; #2进料夹爪松开位标志[0000.11]
ORLD
ANDLD
ORLD
ANDLD
ANDNOT 15.01  ; 扫码NG拉带电机启动
ANDNOT W1.15  ; 有料记忆异常屏蔽（手动调试）
TIMX(550) 0378 D21  ; 报警长延时, 扫码NG放料位有料记忆报警延时
LD TR0
LD T0378  ; 扫码NG放料位有料记忆报警延时
OR W417.06  ; 扫码NG放料位有料记忆[alm]
ANDLD
ANDNOT 200.04  ; 报警清除
OUT W417.06  ; 扫码NG放料位有料记忆[alm]
LD TR0
LD 806.11  ; 氦检NG放料#1位有料感应标志[0006.11]
LD 806.12  ; 氦检NG放料#2位有料感应标志[0006.12]
OR P_On
ANDLD
ANDNOT H17.00  ; 氦检NG放料位有料记忆
LDNOT 806.11  ; 氦检NG放料#1位有料感应标志[0006.11]
ANDNOT 806.12  ; 氦检NG放料#2位有料感应标志[0006.12]
AND H17.00  ; 氦检NG放料位有料记忆
ORLD
ANDLD
LD 853.03  ; 出料伺服Z轴待机位标志
LDNOT 853.03  ; 出料伺服Z轴待机位标志
LDNOT 852.07  ; 出料伺服X轴#1夹爪氦检NG放料位标志
ANDNOT 852.08  ; 出料伺服X轴#2夹爪氦检NG放料位标志
LD 852.03  ; 出料伺服X轴放料位标志
OR 852.04  ; 出料伺服X轴#1腔取料位标志
OR 852.05  ; 出料伺服X轴#2腔取料位标志
OR 852.06  ; 出料伺服X轴#3腔取料位标志
OR 852.09  ; 出料伺服X轴#1夹爪配对取放料位标志
OR 852.10  ; 出料伺服X轴#2夹爪配对取放料位标志
ANDLD
LD 852.07  ; 出料伺服X轴#1夹爪氦检NG放料位标志
AND 853.08  ; 出料伺服Z轴#1夹爪氦检NG放料位标志
AND 800.15  ; #1出料夹爪松开位标志[0000.15]
ORLD
LD 852.08  ; 出料伺服X轴#2夹爪氦检NG放料位标志
AND 853.09  ; 出料伺服Z轴#2夹爪氦检NG放料位标志
AND 801.01  ; #2出料夹爪松开位标志[0001.01]
ORLD
ANDLD
ORLD
ANDLD
ANDNOT 15.02  ; 氦检NG拉带电机启动
ANDNOT W1.15  ; 有料记忆异常屏蔽（手动调试）
TIMX(550) 0379 D21  ; 报警长延时, 氦检NG拉带下料位有料记忆报警延时
LD TR0
LD T0379  ; 氦检NG拉带下料位有料记忆报警延时
OR W417.07  ; 氦检NG拉带下料位有料记忆[alm]
ANDLD
ANDNOT 200.04  ; 报警清除
OUT W417.07  ; 氦检NG拉带下料位有料记忆[alm]

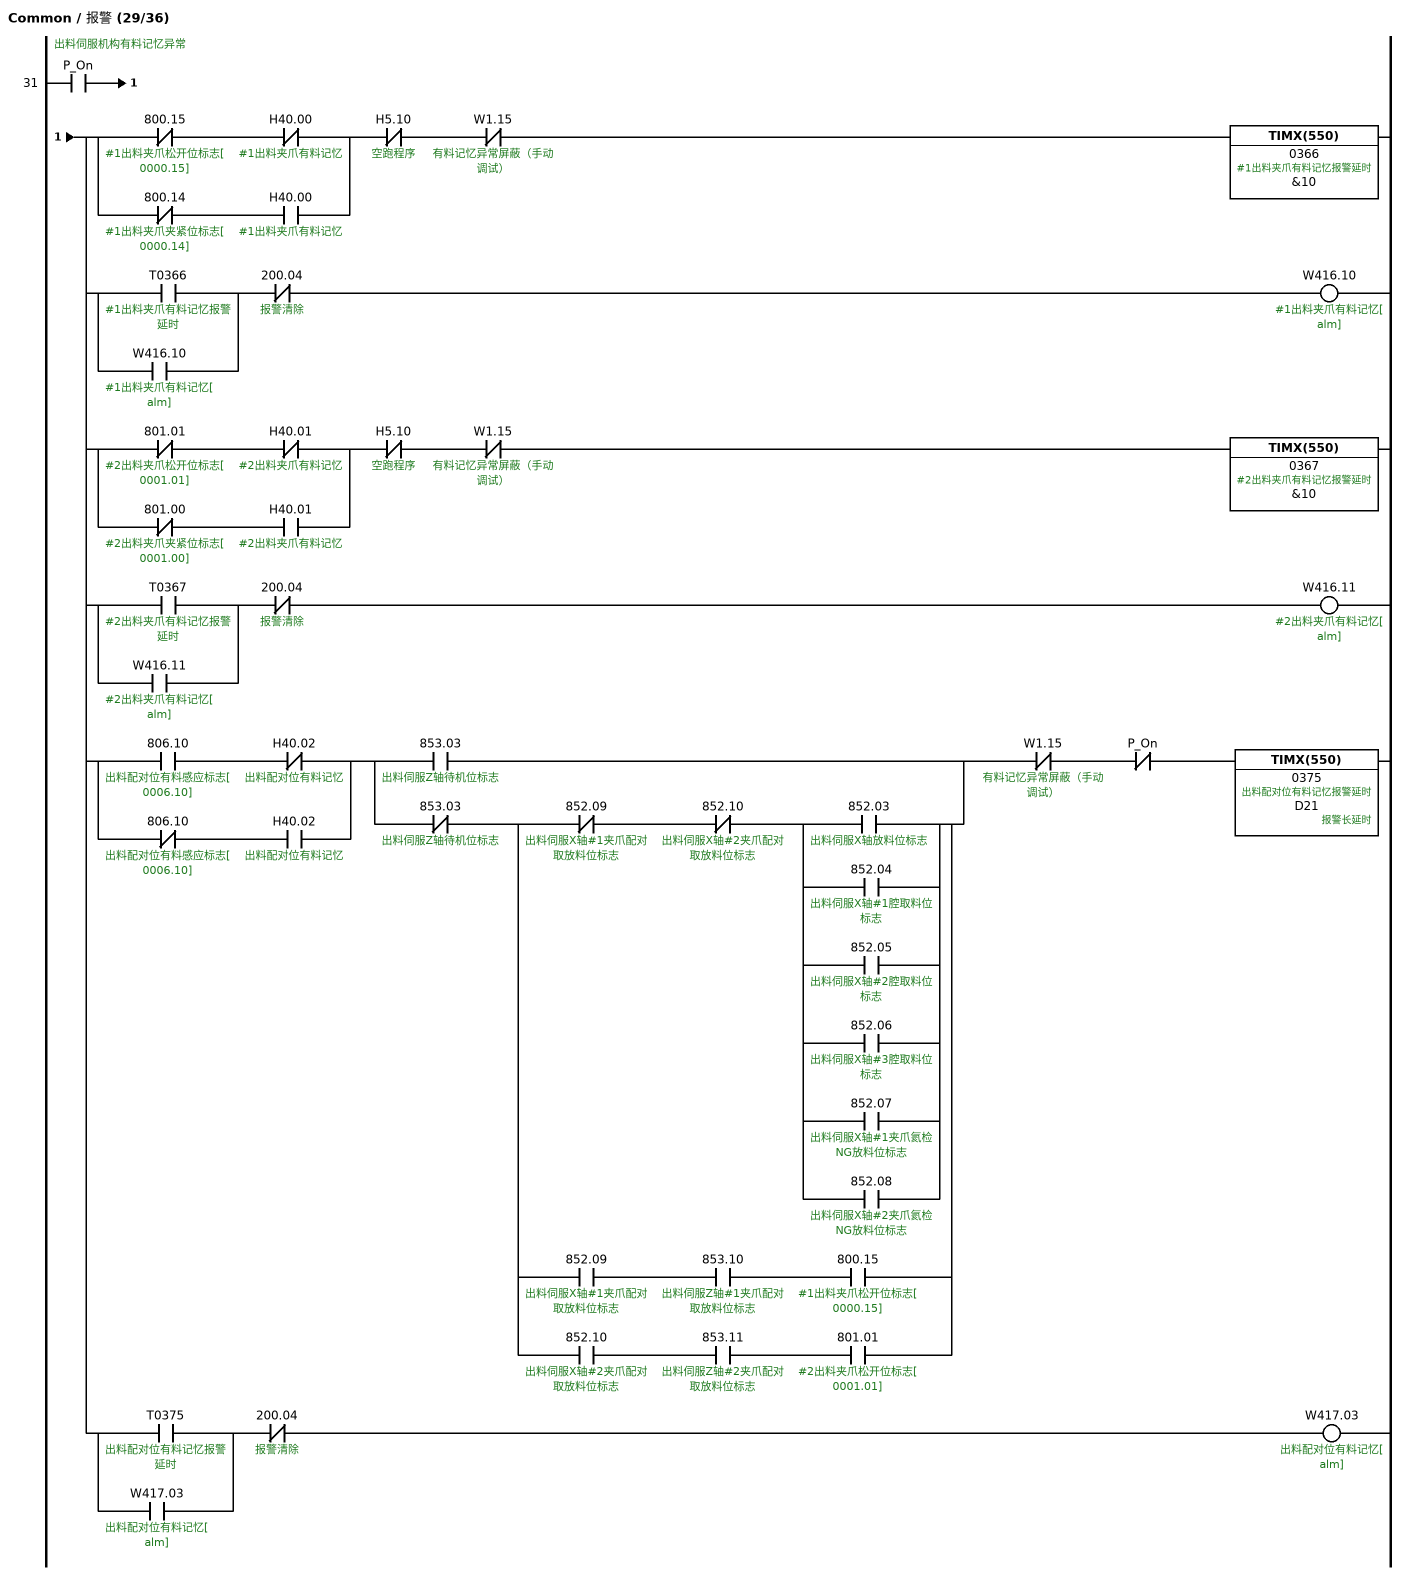
; rung 31: 出料伺服机构有料记忆异常
LD P_On
OUT TR0
LDNOT 800.15  ; #1出料夹爪松开位标志[0000.15]
ANDNOT H40.00  ; #1出料夹爪有料记忆
LDNOT 800.14  ; #1出料夹爪夹紧位标志[0000.14]
AND H40.00  ; #1出料夹爪有料记忆
ORLD
ANDLD
ANDNOT H5.10  ; 空跑程序
ANDNOT W1.15  ; 有料记忆异常屏蔽（手动调试）
TIMX(550) 0366 &10  ; #1出料夹爪有料记忆报警延时
LD TR0
LD T0366  ; #1出料夹爪有料记忆报警延时
OR W416.10  ; #1出料夹爪有料记忆[alm]
ANDLD
ANDNOT 200.04  ; 报警清除
OUT W416.10  ; #1出料夹爪有料记忆[alm]
LD TR0
LDNOT 801.01  ; #2出料夹爪松开位标志[0001.01]
ANDNOT H40.01  ; #2出料夹爪有料记忆
LDNOT 801.00  ; #2出料夹爪夹紧位标志[0001.00]
AND H40.01  ; #2出料夹爪有料记忆
ORLD
ANDLD
ANDNOT H5.10  ; 空跑程序
ANDNOT W1.15  ; 有料记忆异常屏蔽（手动调试）
TIMX(550) 0367 &10  ; #2出料夹爪有料记忆报警延时
LD TR0
LD T0367  ; #2出料夹爪有料记忆报警延时
OR W416.11  ; #2出料夹爪有料记忆[alm]
ANDLD
ANDNOT 200.04  ; 报警清除
OUT W416.11  ; #2出料夹爪有料记忆[alm]
LD TR0
LD 806.10  ; 出料配对位有料感应标志[0006.10]
ANDNOT H40.02  ; 出料配对位有料记忆
LDNOT 806.10  ; 出料配对位有料感应标志[0006.10]
AND H40.02  ; 出料配对位有料记忆
ORLD
ANDLD
LD 853.03  ; 出料伺服Z轴待机位标志
LDNOT 853.03  ; 出料伺服Z轴待机位标志
LDNOT 852.09  ; 出料伺服X轴#1夹爪配对取放料位标志
ANDNOT 852.10  ; 出料伺服X轴#2夹爪配对取放料位标志
LD 852.03  ; 出料伺服X轴放料位标志
OR 852.04  ; 出料伺服X轴#1腔取料位标志
OR 852.05  ; 出料伺服X轴#2腔取料位标志
OR 852.06  ; 出料伺服X轴#3腔取料位标志
OR 852.07  ; 出料伺服X轴#1夹爪氦检NG放料位标志
OR 852.08  ; 出料伺服X轴#2夹爪氦检NG放料位标志
ANDLD
LD 852.09  ; 出料伺服X轴#1夹爪配对取放料位标志
AND 853.10  ; 出料伺服Z轴#1夹爪配对取放料位标志
AND 800.15  ; #1出料夹爪松开位标志[0000.15]
ORLD
LD 852.10  ; 出料伺服X轴#2夹爪配对取放料位标志
AND 853.11  ; 出料伺服Z轴#2夹爪配对取放料位标志
AND 801.01  ; #2出料夹爪松开位标志[0001.01]
ORLD
ANDLD
ORLD
ANDLD
ANDNOT W1.15  ; 有料记忆异常屏蔽（手动调试）
ANDNOT P_On
TIMX(550) 0375 D21  ; 报警长延时, 出料配对位有料记忆报警延时
LD TR0
LD T0375  ; 出料配对位有料记忆报警延时
OR W417.03  ; 出料配对位有料记忆[alm]
ANDLD
ANDNOT 200.04  ; 报警清除
OUT W417.03  ; 出料配对位有料记忆[alm]

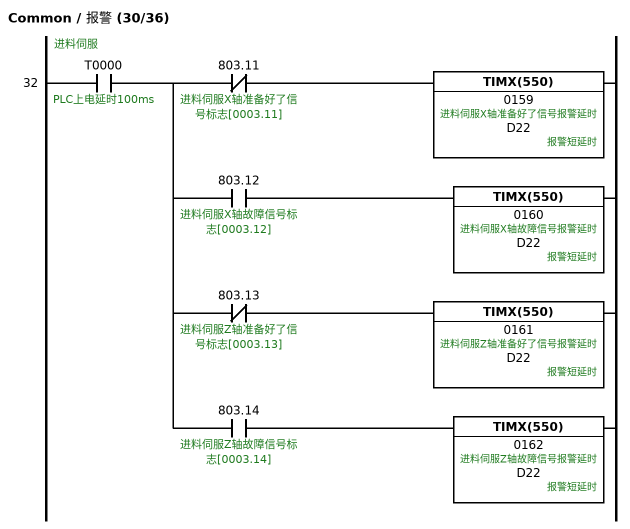
; rung 32: 进料伺服
LD T0000  ; PLC上电延时100ms
OUT TR0
ANDNOT 803.11  ; 进料伺服X轴准备好了信号标志[0003.11]
TIMX(550) 0159 D22  ; 报警短延时, 进料伺服X轴准备好了信号报警延时
LD TR0
AND 803.12  ; 进料伺服X轴故障信号标志[0003.12]
TIMX(550) 0160 D22  ; 报警短延时, 进料伺服X轴故障信号报警延时
LD TR0
ANDNOT 803.13  ; 进料伺服Z轴准备好了信号标志[0003.13]
TIMX(550) 0161 D22  ; 报警短延时, 进料伺服Z轴准备好了信号报警延时
LD TR0
AND 803.14  ; 进料伺服Z轴故障信号标志[0003.14]
TIMX(550) 0162 D22  ; 报警短延时, 进料伺服Z轴故障信号报警延时

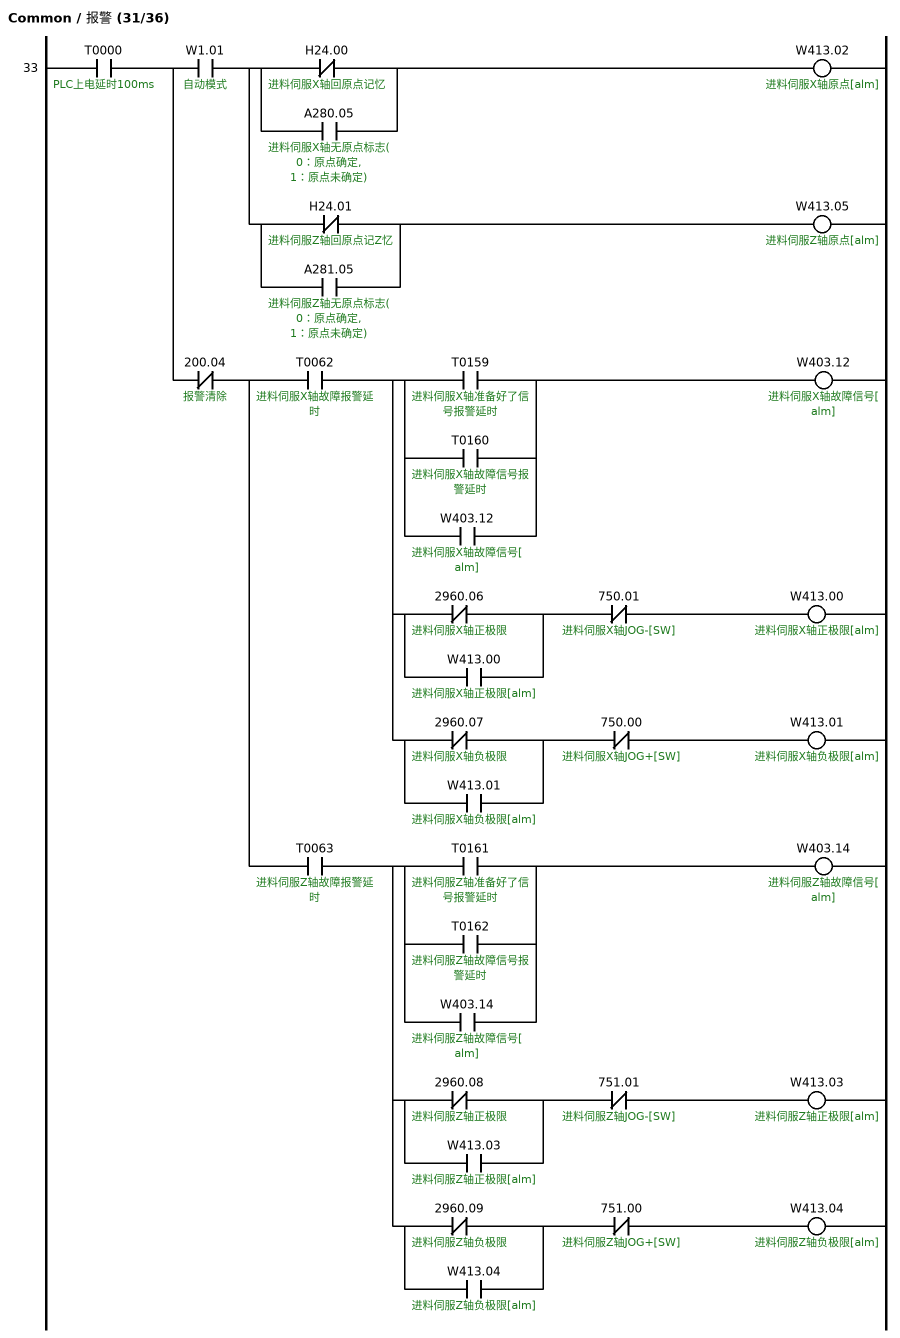
; rung 33
LD T0000  ; PLC上电延时100ms
OUT TR0
AND W1.01  ; 自动模式
OUT TR1
LDNOT H24.00  ; 进料伺服X轴回原点记忆
OR A280.05  ; 进料伺服X轴无原点标志(0：原点确定,1：原点未确定)
ANDLD
OUT W413.02  ; 进料伺服X轴原点[alm]
LD TR1
LDNOT H24.01  ; 进料伺服Z轴回原点记Z忆
OR A281.05  ; 进料伺服Z轴无原点标志(0：原点确定,1：原点未确定)
ANDLD
OUT W413.05  ; 进料伺服Z轴原点[alm]
LD TR0
ANDNOT 200.04  ; 报警清除
OUT TR0
AND T0062  ; 进料伺服X轴故障报警延时
OUT TR1
LD T0159  ; 进料伺服X轴准备好了信号报警延时
OR T0160  ; 进料伺服X轴故障信号报警延时
OR W403.12  ; 进料伺服X轴故障信号[alm]
ANDLD
OUT W403.12  ; 进料伺服X轴故障信号[alm]
LD TR1
LDNOT 2960.06  ; 进料伺服X轴正极限
OR W413.00  ; 进料伺服X轴正极限[alm]
ANDLD
ANDNOT 750.01  ; 进料伺服X轴JOG-[SW]
OUT W413.00  ; 进料伺服X轴正极限[alm]
LD TR1
LDNOT 2960.07  ; 进料伺服X轴负极限
OR W413.01  ; 进料伺服X轴负极限[alm]
ANDLD
ANDNOT 750.00  ; 进料伺服X轴JOG+[SW]
OUT W413.01  ; 进料伺服X轴负极限[alm]
LD TR0
AND T0063  ; 进料伺服Z轴故障报警延时
OUT TR0
LD T0161  ; 进料伺服Z轴准备好了信号报警延时
OR T0162  ; 进料伺服Z轴故障信号报警延时
OR W403.14  ; 进料伺服Z轴故障信号[alm]
ANDLD
OUT W403.14  ; 进料伺服Z轴故障信号[alm]
LD TR0
LDNOT 2960.08  ; 进料伺服Z轴正极限
OR W413.03  ; 进料伺服Z轴正极限[alm]
ANDLD
ANDNOT 751.01  ; 进料伺服Z轴JOG-[SW]
OUT W413.03  ; 进料伺服Z轴正极限[alm]
LD TR0
LDNOT 2960.09  ; 进料伺服Z轴负极限
OR W413.04  ; 进料伺服Z轴负极限[alm]
ANDLD
ANDNOT 751.00  ; 进料伺服Z轴JOG+[SW]
OUT W413.04  ; 进料伺服Z轴负极限[alm]

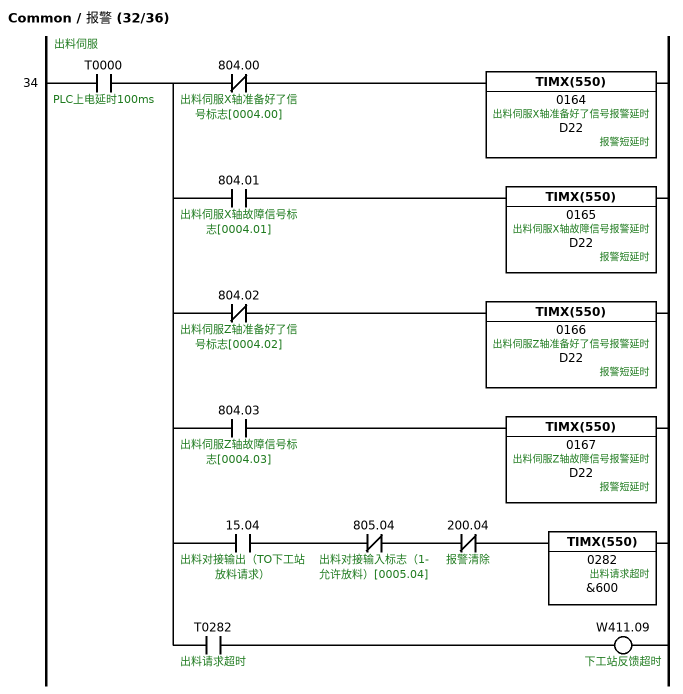
; rung 34: 出料伺服
LD T0000  ; PLC上电延时100ms
OUT TR0
ANDNOT 804.00  ; 出料伺服X轴准备好了信号标志[0004.00]
TIMX(550) 0164 D22  ; 报警短延时, 出料伺服X轴准备好了信号报警延时
LD TR0
AND 804.01  ; 出料伺服X轴故障信号标志[0004.01]
TIMX(550) 0165 D22  ; 报警短延时, 出料伺服X轴故障信号报警延时
LD TR0
ANDNOT 804.02  ; 出料伺服Z轴准备好了信号标志[0004.02]
TIMX(550) 0166 D22  ; 报警短延时, 出料伺服Z轴准备好了信号报警延时
LD TR0
AND 804.03  ; 出料伺服Z轴故障信号标志[0004.03]
TIMX(550) 0167 D22  ; 报警短延时, 出料伺服Z轴故障信号报警延时
LD TR0
AND 15.04  ; 出料对接输出（TO下工站放料请求）
ANDNOT 805.04  ; 出料对接输入标志（1-允许放料）[0005.04]
ANDNOT 200.04  ; 报警清除
TIMX(550) 0282 &600  ; 出料请求超时
LD TR0
AND T0282  ; 出料请求超时
OUT W411.09  ; 下工站反馈超时

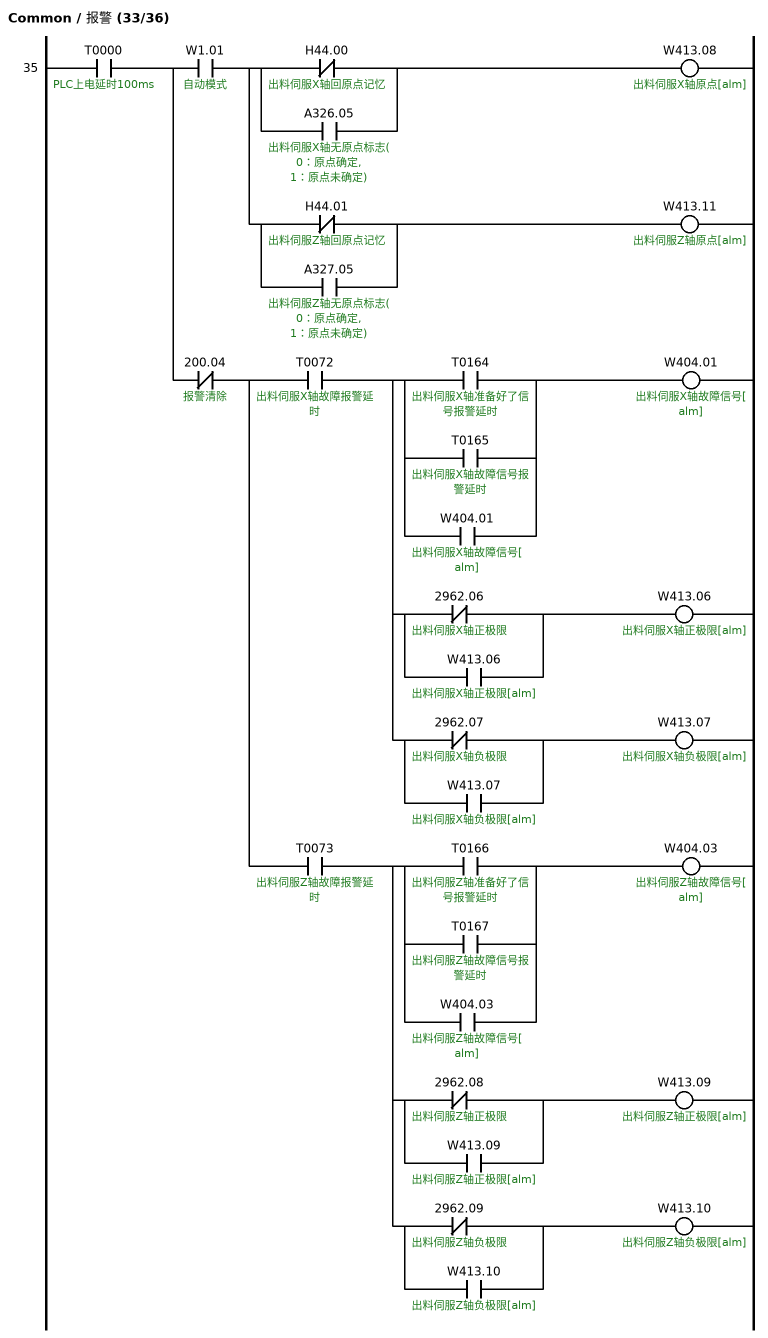
; rung 35
LD T0000  ; PLC上电延时100ms
OUT TR0
AND W1.01  ; 自动模式
OUT TR1
LDNOT H44.00  ; 出料伺服X轴回原点记忆
OR A326.05  ; 出料伺服X轴无原点标志(0：原点确定,1：原点未确定)
ANDLD
OUT W413.08  ; 出料伺服X轴原点[alm]
LD TR1
LDNOT H44.01  ; 出料伺服Z轴回原点记忆
OR A327.05  ; 出料伺服Z轴无原点标志(0：原点确定,1：原点未确定)
ANDLD
OUT W413.11  ; 出料伺服Z轴原点[alm]
LD TR0
ANDNOT 200.04  ; 报警清除
OUT TR0
AND T0072  ; 出料伺服X轴故障报警延时
OUT TR1
LD T0164  ; 出料伺服X轴准备好了信号报警延时
OR T0165  ; 出料伺服X轴故障信号报警延时
OR W404.01  ; 出料伺服X轴故障信号[alm]
ANDLD
OUT W404.01  ; 出料伺服X轴故障信号[alm]
LD TR1
LDNOT 2962.06  ; 出料伺服X轴正极限
OR W413.06  ; 出料伺服X轴正极限[alm]
ANDLD
OUT W413.06  ; 出料伺服X轴正极限[alm]
LD TR1
LDNOT 2962.07  ; 出料伺服X轴负极限
OR W413.07  ; 出料伺服X轴负极限[alm]
ANDLD
OUT W413.07  ; 出料伺服X轴负极限[alm]
LD TR0
AND T0073  ; 出料伺服Z轴故障报警延时
OUT TR0
LD T0166  ; 出料伺服Z轴准备好了信号报警延时
OR T0167  ; 出料伺服Z轴故障信号报警延时
OR W404.03  ; 出料伺服Z轴故障信号[alm]
ANDLD
OUT W404.03  ; 出料伺服Z轴故障信号[alm]
LD TR0
LDNOT 2962.08  ; 出料伺服Z轴正极限
OR W413.09  ; 出料伺服Z轴正极限[alm]
ANDLD
OUT W413.09  ; 出料伺服Z轴正极限[alm]
LD TR0
LDNOT 2962.09  ; 出料伺服Z轴负极限
OR W413.10  ; 出料伺服Z轴负极限[alm]
ANDLD
OUT W413.10  ; 出料伺服Z轴负极限[alm]

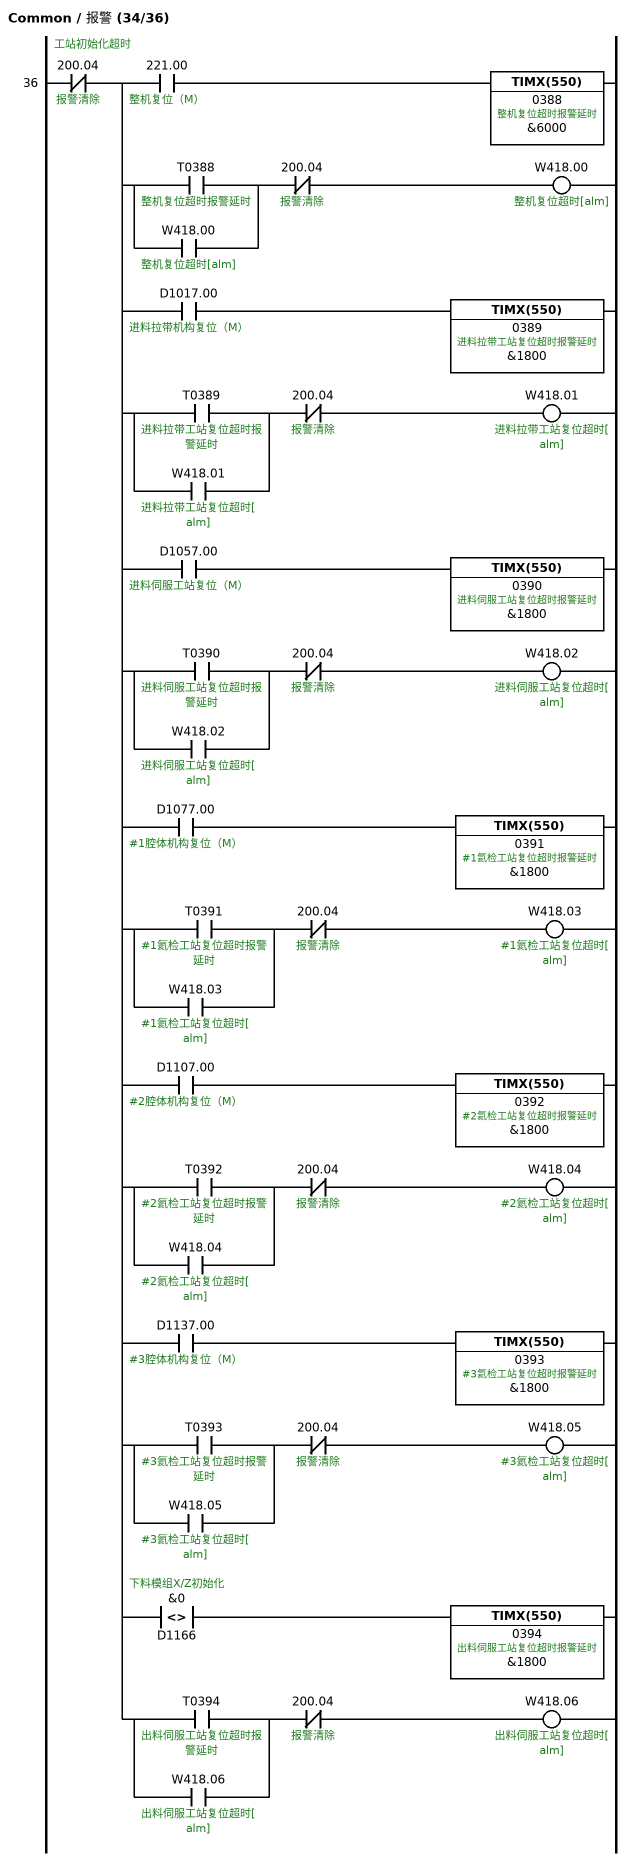
; rung 36: 工站初始化超时
LDNOT 200.04  ; 报警清除
OUT TR0
AND 221.00  ; 整机复位（M）
TIMX(550) 0388 &6000  ; 整机复位超时报警延时
LD TR0
LD T0388  ; 整机复位超时报警延时
OR W418.00  ; 整机复位超时[alm]
ANDLD
ANDNOT 200.04  ; 报警清除
OUT W418.00  ; 整机复位超时[alm]
LD TR0
AND D1017.00  ; 进料拉带机构复位（M）
TIMX(550) 0389 &1800  ; 进料拉带工站复位超时报警延时
LD TR0
LD T0389  ; 进料拉带工站复位超时报警延时
OR W418.01  ; 进料拉带工站复位超时[alm]
ANDLD
ANDNOT 200.04  ; 报警清除
OUT W418.01  ; 进料拉带工站复位超时[alm]
LD TR0
AND D1057.00  ; 进料伺服工站复位（M）
TIMX(550) 0390 &1800  ; 进料伺服工站复位超时报警延时
LD TR0
LD T0390  ; 进料伺服工站复位超时报警延时
OR W418.02  ; 进料伺服工站复位超时[alm]
ANDLD
ANDNOT 200.04  ; 报警清除
OUT W418.02  ; 进料伺服工站复位超时[alm]
LD TR0
AND D1077.00  ; #1腔体机构复位（M）
TIMX(550) 0391 &1800  ; #1氦检工站复位超时报警延时
LD TR0
LD T0391  ; #1氦检工站复位超时报警延时
OR W418.03  ; #1氦检工站复位超时[alm]
ANDLD
ANDNOT 200.04  ; 报警清除
OUT W418.03  ; #1氦检工站复位超时[alm]
LD TR0
AND D1107.00  ; #2腔体机构复位（M）
TIMX(550) 0392 &1800  ; #2氦检工站复位超时报警延时
LD TR0
LD T0392  ; #2氦检工站复位超时报警延时
OR W418.04  ; #2氦检工站复位超时[alm]
ANDLD
ANDNOT 200.04  ; 报警清除
OUT W418.04  ; #2氦检工站复位超时[alm]
LD TR0
AND D1137.00  ; #3腔体机构复位（M）
TIMX(550) 0393 &1800  ; #3氦检工站复位超时报警延时
LD TR0
LD T0393  ; #3氦检工站复位超时报警延时
OR W418.05  ; #3氦检工站复位超时[alm]
ANDLD
ANDNOT 200.04  ; 报警清除
OUT W418.05  ; #3氦检工站复位超时[alm]
LD TR0
AND<>(305) &0 D1166  ; 下料模组X/Z初始化
TIMX(550) 0394 &1800  ; 出料伺服工站复位超时报警延时
LD TR0
LD T0394  ; 出料伺服工站复位超时报警延时
OR W418.06  ; 出料伺服工站复位超时[alm]
ANDLD
ANDNOT 200.04  ; 报警清除
OUT W418.06  ; 出料伺服工站复位超时[alm]

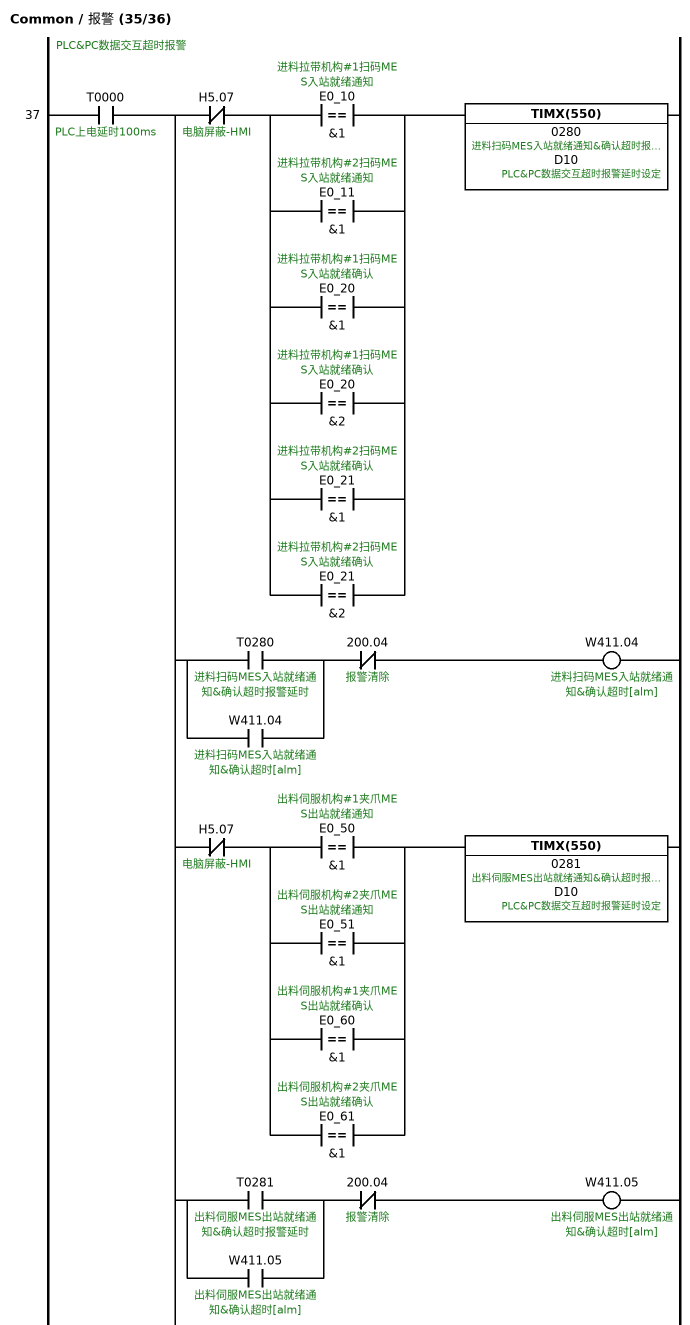

